gfCNCPoint3[28774] = {X 352.3341, Y -3.5325, Z 11.0000, A 0.000, B 0.000, C 0.000 }
gfCNCPoint3[28775] = {X 352.3341, Y -3.5325, Z -1.6667, A 0.000, B 0.000, C 0.000 }
gfCNCPoint3[28776] = {X 352.3341, Y -3.5325, Z -4.6667, A 0.000, B 0.000, C 0.000 }
gfCNCPoint3[28777] = {X 351.5863, Y 0.4784, Z -4.6667, A 0.000, B 0.000, C 0.000 }
gfCNCPoint3[28778] = {X 351.8700, Y 0.5313, Z -4.6667, A 0.000, B 0.000, C 0.000 }
gfCNCPoint3[28779] = {X 353.8050, Y 1.0172, Z -4.6667, A 0.000, B 0.000, C 0.000 }
gfCNCPoint3[28780] = {X 355.6853, Y 1.6845, Z -4.6667, A 0.000, B 0.000, C 0.000 }
gfCNCPoint3[28781] = {X 357.4938, Y 2.5269, Z -4.6667, A 0.000, B 0.000, C 0.000 }
gfCNCPoint3[28782] = {X 359.2143, Y 3.5371, Z -4.6667, A 0.000, B 0.000, C 0.000 }
gfCNCPoint3[28783] = {X 360.8312, Y 4.7058, Z -4.6667, A 0.000, B 0.000, C 0.000 }
gfCNCPoint3[28784] = {X 362.3301, Y 6.0226, Z -4.6667, A 0.000, B 0.000, C 0.000 }
gfCNCPoint3[28785] = {X 363.6974, Y 7.4756, Z -4.6667, A 0.000, B 0.000, C 0.000 }
gfCNCPoint3[28786] = {X 365.1619, Y 9.3656, Z -4.6667, A 0.000, B 0.000, C 0.000 }
gfCNCPoint3[28787] = {X 366.4369, Y 11.3883, Z -4.6667, A 0.000, B 0.000, C 0.000 }
gfCNCPoint3[28788] = {X 367.5105, Y 13.5247, Z -4.6667, A 0.000, B 0.000, C 0.000 }
gfCNCPoint3[28789] = {X 368.3726, Y 15.7549, Z -4.6667, A 0.000, B 0.000, C 0.000 }
gfCNCPoint3[28790] = {X 369.0153, Y 18.0579, Z -4.6667, A 0.000, B 0.000, C 0.000 }
gfCNCPoint3[28791] = {X 369.4989, Y 20.6961, Z -4.6667, A 0.000, B 0.000, C 0.000 }
gfCNCPoint3[28792] = {X 369.7571, Y 23.3657, Z -4.6667, A 0.000, B 0.000, C 0.000 }
gfCNCPoint3[28793] = {X 369.7880, Y 26.0477, Z -4.6667, A 0.000, B 0.000, C 0.000 }
gfCNCPoint3[28794] = {X 369.5915, Y 28.7226, Z -4.6667, A 0.000, B 0.000, C 0.000 }
gfCNCPoint3[28795] = {X 369.1690, Y 31.3712, Z -4.6667, A 0.000, B 0.000, C 0.000 }
gfCNCPoint3[28796] = {X 368.6451, Y 33.4755, Z -4.6667, A 0.000, B 0.000, C 0.000 }
gfCNCPoint3[28797] = {X 367.9373, Y 35.5252, Z -4.6667, A 0.000, B 0.000, C 0.000 }
gfCNCPoint3[28798] = {X 367.0512, Y 37.5044, Z -4.6667, A 0.000, B 0.000, C 0.000 }
gfCNCPoint3[28799] = {X 365.9938, Y 39.3976, Z -4.6667, A 0.000, B 0.000, C 0.000 }
gfCNCPoint3[28800] = {X 364.7733, Y 41.1900, Z -4.6667, A 0.000, B 0.000, C 0.000 }
gfCNCPoint3[28801] = {X 364.6545, Y 41.3528, Z -4.6667, A 0.000, B 0.000, C 0.000 }
gfCNCPoint3[28802] = {X 364.0247, Y 42.1261, Z -4.6667, A 0.000, B 0.000, C 0.000 }
gfCNCPoint3[28803] = {X 362.7636, Y 43.5412, Z -4.6667, A 0.000, B 0.000, C 0.000 }
gfCNCPoint3[28804] = {X 361.3817, Y 44.8384, Z -4.6667, A 0.000, B 0.000, C 0.000 }
gfCNCPoint3[28805] = {X 359.8899, Y 46.0077, Z -4.6667, A 0.000, B 0.000, C 0.000 }
gfCNCPoint3[28806] = {X 358.3000, Y 47.0398, Z -4.6667, A 0.000, B 0.000, C 0.000 }
gfCNCPoint3[28807] = {X 356.6247, Y 47.9264, Z -4.6667, A 0.000, B 0.000, C 0.000 }
gfCNCPoint3[28808] = {X 356.2232, Y 48.1165, Z -4.6667, A 0.000, B 0.000, C 0.000 }
gfCNCPoint3[28809] = {X 354.0252, Y 48.9371, Z -4.6667, A 0.000, B 0.000, C 0.000 }
gfCNCPoint3[28810] = {X 351.7551, Y 49.5298, Z -4.6667, A 0.000, B 0.000, C 0.000 }
gfCNCPoint3[28811] = {X 349.4364, Y 49.8883, Z -4.6667, A 0.000, B 0.000, C 0.000 }
gfCNCPoint3[28812] = {X 347.0933, Y 50.0089, Z -4.6667, A 0.000, B 0.000, C 0.000 }
gfCNCPoint3[28813] = {X 345.0267, Y 49.9741, Z -4.6667, A 0.000, B 0.000, C 0.000 }
gfCNCPoint3[28814] = {X 342.9709, Y 49.7601, Z -4.6667, A 0.000, B 0.000, C 0.000 }
gfCNCPoint3[28815] = {X 340.9414, Y 49.3687, Z -4.6667, A 0.000, B 0.000, C 0.000 }
gfCNCPoint3[28816] = {X 338.9535, Y 48.8027, Z -4.6667, A 0.000, B 0.000, C 0.000 }
gfCNCPoint3[28817] = {X 337.0223, Y 48.0664, Z -4.6667, A 0.000, B 0.000, C 0.000 }
gfCNCPoint3[28818] = {X 335.1621, Y 47.1654, Z -4.6667, A 0.000, B 0.000, C 0.000 }
gfCNCPoint3[28819] = {X 333.5779, Y 46.1879, Z -4.6667, A 0.000, B 0.000, C 0.000 }
gfCNCPoint3[28820] = {X 332.0749, Y 45.0895, Z -4.6667, A 0.000, B 0.000, C 0.000 }
gfCNCPoint3[28821] = {X 330.6624, Y 43.8770, Z -4.6667, A 0.000, B 0.000, C 0.000 }
gfCNCPoint3[28822] = {X 329.7213, Y 43.8764, Z -4.6667, A 0.000, B 0.000, C 0.000 }
gfCNCPoint3[28823] = {X 328.8027, Y 43.6721, Z -4.6667, A 0.000, B 0.000, C 0.000 }
gfCNCPoint3[28824] = {X 327.9501, Y 43.2738, Z -4.6667, A 0.000, B 0.000, C 0.000 }
gfCNCPoint3[28825] = {X 327.2040, Y 42.7002, Z -4.6667, A 0.000, B 0.000, C 0.000 }
gfCNCPoint3[28826] = {X 326.5808, Y 42.0925, Z -4.6667, A 0.000, B 0.000, C 0.000 }
gfCNCPoint3[28827] = {X 325.9523, Y 41.3190, Z -4.6667, A 0.000, B 0.000, C 0.000 }
gfCNCPoint3[28828] = {X 325.5179, Y 40.4220, Z -4.6667, A 0.000, B 0.000, C 0.000 }
gfCNCPoint3[28829] = {X 325.3006, Y 39.4493, Z -4.6667, A 0.000, B 0.000, C 0.000 }
gfCNCPoint3[28830] = {X 325.3120, Y 38.4527, Z -4.6667, A 0.000, B 0.000, C 0.000 }
gfCNCPoint3[28831] = {X 325.5514, Y 37.4852, Z -4.6667, A 0.000, B 0.000, C 0.000 }
gfCNCPoint3[28832] = {X 326.0062, Y 36.5984, Z -4.6667, A 0.000, B 0.000, C 0.000 }
gfCNCPoint3[28833] = {X 330.2395, Y 30.2687, Z -4.6667, A 0.000, B 0.000, C 0.000 }
gfCNCPoint3[28834] = {X 330.8410, Y 29.5518, Z -4.6667, A 0.000, B 0.000, C 0.000 }
gfCNCPoint3[28835] = {X 331.5827, Y 28.9812, Z -4.6667, A 0.000, B 0.000, C 0.000 }
gfCNCPoint3[28836] = {X 332.4298, Y 28.5837, Z -4.6667, A 0.000, B 0.000, C 0.000 }
gfCNCPoint3[28837] = {X 333.3427, Y 28.3779, Z -4.6667, A 0.000, B 0.000, C 0.000 }
gfCNCPoint3[28838] = {X 334.2785, Y 28.3736, Z -4.6667, A 0.000, B 0.000, C 0.000 }
gfCNCPoint3[28839] = {X 335.1933, Y 28.5709, Z -4.6667, A 0.000, B 0.000, C 0.000 }
gfCNCPoint3[28840] = {X 336.0441, Y 28.9606, Z -4.6667, A 0.000, B 0.000, C 0.000 }
gfCNCPoint3[28841] = {X 336.7910, Y 29.5243, Z -4.6667, A 0.000, B 0.000, C 0.000 }
gfCNCPoint3[28842] = {X 337.4284, Y 30.1382, Z -4.6667, A 0.000, B 0.000, C 0.000 }
gfCNCPoint3[28843] = {X 337.9529, Y 30.7612, Z -4.6667, A 0.000, B 0.000, C 0.000 }
gfCNCPoint3[28844] = {X 338.3512, Y 31.4715, Z -4.6667, A 0.000, B 0.000, C 0.000 }
gfCNCPoint3[28845] = {X 338.6091, Y 32.2439, Z -4.6667, A 0.000, B 0.000, C 0.000 }
gfCNCPoint3[28846] = {X 338.7175, Y 33.0510, Z -4.6667, A 0.000, B 0.000, C 0.000 }
gfCNCPoint3[28847] = {X 338.6725, Y 33.8642, Z -4.6667, A 0.000, B 0.000, C 0.000 }
gfCNCPoint3[28848] = {X 339.4371, Y 34.5550, Z -4.6667, A 0.000, B 0.000, C 0.000 }
gfCNCPoint3[28849] = {X 340.2341, Y 35.2082, Z -4.6667, A 0.000, B 0.000, C 0.000 }
gfCNCPoint3[28850] = {X 341.5315, Y 36.0599, Z -4.6667, A 0.000, B 0.000, C 0.000 }
gfCNCPoint3[28851] = {X 342.9391, Y 36.7134, Z -4.6667, A 0.000, B 0.000, C 0.000 }
gfCNCPoint3[28852] = {X 344.4270, Y 37.1548, Z -4.6667, A 0.000, B 0.000, C 0.000 }
gfCNCPoint3[28853] = {X 345.9633, Y 37.3746, Z -4.6667, A 0.000, B 0.000, C 0.000 }
gfCNCPoint3[28854] = {X 347.5152, Y 37.3683, Z -4.6667, A 0.000, B 0.000, C 0.000 }
gfCNCPoint3[28855] = {X 348.9560, Y 37.1753, Z -4.6667, A 0.000, B 0.000, C 0.000 }
gfCNCPoint3[28856] = {X 350.3462, Y 36.7501, Z -4.6667, A 0.000, B 0.000, C 0.000 }
gfCNCPoint3[28857] = {X 351.6486, Y 36.1043, Z -4.6667, A 0.000, B 0.000, C 0.000 }
gfCNCPoint3[28858] = {X 352.8283, Y 35.2549, Z -4.6667, A 0.000, B 0.000, C 0.000 }
gfCNCPoint3[28859] = {X 353.9821, Y 34.1341, Z -4.6667, A 0.000, B 0.000, C 0.000 }
gfCNCPoint3[28860] = {X 354.9806, Y 32.8730, Z -4.6667, A 0.000, B 0.000, C 0.000 }
gfCNCPoint3[28861] = {X 355.8069, Y 31.4930, Z -4.6667, A 0.000, B 0.000, C 0.000 }
gfCNCPoint3[28862] = {X 356.4470, Y 30.0173, Z -4.6667, A 0.000, B 0.000, C 0.000 }
gfCNCPoint3[28863] = {X 356.8901, Y 28.4711, Z -4.6667, A 0.000, B 0.000, C 0.000 }
gfCNCPoint3[28864] = {X 357.1634, Y 26.7828, Z -4.6667, A 0.000, B 0.000, C 0.000 }
gfCNCPoint3[28865] = {X 357.2747, Y 25.0763, Z -4.6667, A 0.000, B 0.000, C 0.000 }
gfCNCPoint3[28866] = {X 357.2231, Y 23.3669, Z -4.6667, A 0.000, B 0.000, C 0.000 }
gfCNCPoint3[28867] = {X 357.0089, Y 21.6701, Z -4.6667, A 0.000, B 0.000, C 0.000 }
gfCNCPoint3[28868] = {X 356.6550, Y 20.1540, Z -4.6667, A 0.000, B 0.000, C 0.000 }
gfCNCPoint3[28869] = {X 356.1053, Y 18.6975, Z -4.6667, A 0.000, B 0.000, C 0.000 }
gfCNCPoint3[28870] = {X 355.3691, Y 17.3257, Z -4.6667, A 0.000, B 0.000, C 0.000 }
gfCNCPoint3[28871] = {X 354.4594, Y 16.0623, Z -4.6667, A 0.000, B 0.000, C 0.000 }
gfCNCPoint3[28872] = {X 353.5887, Y 15.1354, Z -4.6667, A 0.000, B 0.000, C 0.000 }
gfCNCPoint3[28873] = {X 352.5980, Y 14.3381, Z -4.6667, A 0.000, B 0.000, C 0.000 }
gfCNCPoint3[28874] = {X 351.5062, Y 13.6859, Z -4.6667, A 0.000, B 0.000, C 0.000 }
gfCNCPoint3[28875] = {X 350.3346, Y 13.1914, Z -4.6667, A 0.000, B 0.000, C 0.000 }
gfCNCPoint3[28876] = {X 349.1057, Y 12.8640, Z -4.6667, A 0.000, B 0.000, C 0.000 }
gfCNCPoint3[28877] = {X 347.3453, Y 12.6451, Z -4.6667, A 0.000, B 0.000, C 0.000 }
gfCNCPoint3[28878] = {X 345.5714, Y 12.6609, Z -4.6667, A 0.000, B 0.000, C 0.000 }
gfCNCPoint3[28879] = {X 343.8152, Y 12.9112, Z -4.6667, A 0.000, B 0.000, C 0.000 }
gfCNCPoint3[28880] = {X 342.1076, Y 13.3916, Z -4.6667, A 0.000, B 0.000, C 0.000 }
gfCNCPoint3[28881] = {X 340.4785, Y 14.0937, Z -4.6667, A 0.000, B 0.000, C 0.000 }
gfCNCPoint3[28882] = {X 338.9566, Y 15.0051, Z -4.6667, A 0.000, B 0.000, C 0.000 }
gfCNCPoint3[28883] = {X 338.9177, Y 15.8498, Z -4.6667, A 0.000, B 0.000, C 0.000 }
gfCNCPoint3[28884] = {X 338.7151, Y 16.6708, Z -4.6667, A 0.000, B 0.000, C 0.000 }
gfCNCPoint3[28885] = {X 338.3564, Y 17.4366, Z -4.6667, A 0.000, B 0.000, C 0.000 }
gfCNCPoint3[28886] = {X 337.8553, Y 18.1179, Z -4.6667, A 0.000, B 0.000, C 0.000 }
gfCNCPoint3[28887] = {X 337.2312, Y 18.6884, Z -4.6667, A 0.000, B 0.000, C 0.000 }
gfCNCPoint3[28888] = {X 336.5140, Y 19.2162, Z -4.6667, A 0.000, B 0.000, C 0.000 }
gfCNCPoint3[28889] = {X 335.6982, Y 19.6754, Z -4.6667, A 0.000, B 0.000, C 0.000 }
gfCNCPoint3[28890] = {X 334.8027, Y 19.9480, Z -4.6667, A 0.000, B 0.000, C 0.000 }
gfCNCPoint3[28891] = {X 333.8694, Y 20.0213, Z -4.6667, A 0.000, B 0.000, C 0.000 }
gfCNCPoint3[28892] = {X 332.9422, Y 19.8919, Z -4.6667, A 0.000, B 0.000, C 0.000 }
gfCNCPoint3[28893] = {X 332.0647, Y 19.5657, Z -4.6667, A 0.000, B 0.000, C 0.000 }
gfCNCPoint3[28894] = {X 331.2781, Y 19.0581, Z -4.6667, A 0.000, B 0.000, C 0.000 }
gfCNCPoint3[28895] = {X 330.6193, Y 18.3931, Z -4.6667, A 0.000, B 0.000, C 0.000 }
gfCNCPoint3[28896] = {X 330.1192, Y 17.6017, Z -4.6667, A 0.000, B 0.000, C 0.000 }
gfCNCPoint3[28897] = {X 326.5942, Y 10.3502, Z -4.6667, A 0.000, B 0.000, C 0.000 }
gfCNCPoint3[28898] = {X 326.2930, Y 9.5272, Z -4.6667, A 0.000, B 0.000, C 0.000 }
gfCNCPoint3[28899] = {X 326.1640, Y 8.6602, Z -4.6667, A 0.000, B 0.000, C 0.000 }
gfCNCPoint3[28900] = {X 326.2128, Y 7.7851, Z -4.6667, A 0.000, B 0.000, C 0.000 }
gfCNCPoint3[28901] = {X 326.4371, Y 6.9379, Z -4.6667, A 0.000, B 0.000, C 0.000 }
gfCNCPoint3[28902] = {X 326.8278, Y 6.1534, Z -4.6667, A 0.000, B 0.000, C 0.000 }
gfCNCPoint3[28903] = {X 327.3688, Y 5.4638, Z -4.6667, A 0.000, B 0.000, C 0.000 }
gfCNCPoint3[28904] = {X 328.0379, Y 4.8977, Z -4.6667, A 0.000, B 0.000, C 0.000 }
gfCNCPoint3[28905] = {X 328.7084, Y 4.4386, Z -4.6667, A 0.000, B 0.000, C 0.000 }
gfCNCPoint3[28906] = {X 329.5888, Y 3.9825, Z -4.6667, A 0.000, B 0.000, C 0.000 }
gfCNCPoint3[28907] = {X 330.5501, Y 3.7392, Z -4.6667, A 0.000, B 0.000, C 0.000 }
gfCNCPoint3[28908] = {X 331.5414, Y 3.7215, Z -4.6667, A 0.000, B 0.000, C 0.000 }
gfCNCPoint3[28909] = {X 332.5107, Y 3.9303, Z -4.6667, A 0.000, B 0.000, C 0.000 }
gfCNCPoint3[28910] = {X 333.9976, Y 3.1006, Z -4.6667, A 0.000, B 0.000, C 0.000 }
gfCNCPoint3[28911] = {X 335.5315, Y 2.3616, Z -4.6667, A 0.000, B 0.000, C 0.000 }
gfCNCPoint3[28912] = {X 337.6677, Y 1.4950, Z -4.6667, A 0.000, B 0.000, C 0.000 }
gfCNCPoint3[28913] = {X 339.8716, Y 0.8189, Z -4.6667, A 0.000, B 0.000, C 0.000 }
gfCNCPoint3[28914] = {X 342.1263, Y 0.3386, Z -4.6667, A 0.000, B 0.000, C 0.000 }
gfCNCPoint3[28915] = {X 344.4144, Y 0.0577, Z -4.6667, A 0.000, B 0.000, C 0.000 }
gfCNCPoint3[28916] = {X 346.7183, Y -0.0216, Z -4.6667, A 0.000, B 0.000, C 0.000 }
gfCNCPoint3[28917] = {X 349.0203, Y 0.1013, Z -4.6667, A 0.000, B 0.000, C 0.000 }
gfCNCPoint3[28918] = {X 351.3027, Y 0.4255, Z -4.6667, A 0.000, B 0.000, C 0.000 }
gfCNCPoint3[28919] = {X 351.5863, Y 0.4784, Z -4.6667, A 0.000, B 0.000, C 0.000 }
gfCNCPoint3[28920] = {X 352.3195, Y -3.4539, Z -4.6667, A 0.000, B 0.000, C 0.000 }
gfCNCPoint3[28921] = {X 351.5717, Y 0.5570, Z -4.6667, A 0.000, B 0.000, C 0.000 }
gfCNCPoint3[28922] = {X 351.8548, Y 0.6098, Z -4.6667, A 0.000, B 0.000, C 0.000 }
gfCNCPoint3[28923] = {X 353.7823, Y 1.0939, Z -4.6667, A 0.000, B 0.000, C 0.000 }
gfCNCPoint3[28924] = {X 355.6553, Y 1.7586, Z -4.6667, A 0.000, B 0.000, C 0.000 }
gfCNCPoint3[28925] = {X 357.4569, Y 2.5979, Z -4.6667, A 0.000, B 0.000, C 0.000 }
gfCNCPoint3[28926] = {X 359.1708, Y 3.6042, Z -4.6667, A 0.000, B 0.000, C 0.000 }
gfCNCPoint3[28927] = {X 360.7815, Y 4.7685, Z -4.6667, A 0.000, B 0.000, C 0.000 }
gfCNCPoint3[28928] = {X 362.2746, Y 6.0802, Z -4.6667, A 0.000, B 0.000, C 0.000 }
gfCNCPoint3[28929] = {X 363.6366, Y 7.5276, Z -4.6667, A 0.000, B 0.000, C 0.000 }
gfCNCPoint3[28930] = {X 365.0963, Y 9.4115, Z -4.6667, A 0.000, B 0.000, C 0.000 }
gfCNCPoint3[28931] = {X 366.3672, Y 11.4276, Z -4.6667, A 0.000, B 0.000, C 0.000 }
gfCNCPoint3[28932] = {X 367.4374, Y 13.5571, Z -4.6667, A 0.000, B 0.000, C 0.000 }
gfCNCPoint3[28933] = {X 368.2967, Y 15.7801, Z -4.6667, A 0.000, B 0.000, C 0.000 }
gfCNCPoint3[28934] = {X 368.9373, Y 18.0757, Z -4.6667, A 0.000, B 0.000, C 0.000 }
gfCNCPoint3[28935] = {X 369.4196, Y 20.7071, Z -4.6667, A 0.000, B 0.000, C 0.000 }
gfCNCPoint3[28936] = {X 369.6772, Y 23.3700, Z -4.6667, A 0.000, B 0.000, C 0.000 }
gfCNCPoint3[28937] = {X 369.7081, Y 26.0452, Z -4.6667, A 0.000, B 0.000, C 0.000 }
gfCNCPoint3[28938] = {X 369.5121, Y 28.7133, Z -4.6667, A 0.000, B 0.000, C 0.000 }
gfCNCPoint3[28939] = {X 369.0906, Y 31.3552, Z -4.6667, A 0.000, B 0.000, C 0.000 }
gfCNCPoint3[28940] = {X 368.5684, Y 33.4527, Z -4.6667, A 0.000, B 0.000, C 0.000 }
gfCNCPoint3[28941] = {X 367.8629, Y 35.4959, Z -4.6667, A 0.000, B 0.000, C 0.000 }
gfCNCPoint3[28942] = {X 366.9796, Y 37.4688, Z -4.6667, A 0.000, B 0.000, C 0.000 }
gfCNCPoint3[28943] = {X 365.9256, Y 39.3559, Z -4.6667, A 0.000, B 0.000, C 0.000 }
gfCNCPoint3[28944] = {X 364.7089, Y 41.1425, Z -4.6667, A 0.000, B 0.000, C 0.000 }
gfCNCPoint3[28945] = {X 364.5911, Y 41.3039, Z -4.6667, A 0.000, B 0.000, C 0.000 }
gfCNCPoint3[28946] = {X 363.9627, Y 42.0756, Z -4.6667, A 0.000, B 0.000, C 0.000 }
gfCNCPoint3[28947] = {X 362.7063, Y 43.4853, Z -4.6667, A 0.000, B 0.000, C 0.000 }
gfCNCPoint3[28948] = {X 361.3296, Y 44.7777, Z -4.6667, A 0.000, B 0.000, C 0.000 }
gfCNCPoint3[28949] = {X 359.8434, Y 45.9426, Z -4.6667, A 0.000, B 0.000, C 0.000 }
gfCNCPoint3[28950] = {X 358.2595, Y 46.9708, Z -4.6667, A 0.000, B 0.000, C 0.000 }
gfCNCPoint3[28951] = {X 356.5905, Y 47.8541, Z -4.6667, A 0.000, B 0.000, C 0.000 }
gfCNCPoint3[28952] = {X 356.1902, Y 48.0436, Z -4.6667, A 0.000, B 0.000, C 0.000 }
gfCNCPoint3[28953] = {X 353.9998, Y 48.8612, Z -4.6667, A 0.000, B 0.000, C 0.000 }
gfCNCPoint3[28954] = {X 351.7376, Y 49.4517, Z -4.6667, A 0.000, B 0.000, C 0.000 }
gfCNCPoint3[28955] = {X 349.4271, Y 49.8088, Z -4.6667, A 0.000, B 0.000, C 0.000 }
gfCNCPoint3[28956] = {X 347.0922, Y 49.9289, Z -4.6667, A 0.000, B 0.000, C 0.000 }
gfCNCPoint3[28957] = {X 345.0325, Y 49.8943, Z -4.6667, A 0.000, B 0.000, C 0.000 }
gfCNCPoint3[28958] = {X 342.9836, Y 49.6811, Z -4.6667, A 0.000, B 0.000, C 0.000 }
gfCNCPoint3[28959] = {X 340.9608, Y 49.2911, Z -4.6667, A 0.000, B 0.000, C 0.000 }
gfCNCPoint3[28960] = {X 338.9796, Y 48.7270, Z -4.6667, A 0.000, B 0.000, C 0.000 }
gfCNCPoint3[28961] = {X 337.0547, Y 47.9933, Z -4.6667, A 0.000, B 0.000, C 0.000 }
gfCNCPoint3[28962] = {X 335.2008, Y 47.0953, Z -4.6667, A 0.000, B 0.000, C 0.000 }
gfCNCPoint3[28963] = {X 333.6119, Y 46.1143, Z -4.6667, A 0.000, B 0.000, C 0.000 }
gfCNCPoint3[28964] = {X 332.1052, Y 45.0114, Z -4.6667, A 0.000, B 0.000, C 0.000 }
gfCNCPoint3[28965] = {X 330.6899, Y 43.7933, Z -4.6667, A 0.000, B 0.000, C 0.000 }
gfCNCPoint3[28966] = {X 329.7572, Y 43.7998, Z -4.6667, A 0.000, B 0.000, C 0.000 }
gfCNCPoint3[28967] = {X 328.8457, Y 43.6022, Z -4.6667, A 0.000, B 0.000, C 0.000 }
gfCNCPoint3[28968] = {X 327.9994, Y 43.2101, Z -4.6667, A 0.000, B 0.000, C 0.000 }
gfCNCPoint3[28969] = {X 327.2594, Y 42.6425, Z -4.6667, A 0.000, B 0.000, C 0.000 }
gfCNCPoint3[28970] = {X 326.6366, Y 42.0352, Z -4.6667, A 0.000, B 0.000, C 0.000 }
gfCNCPoint3[28971] = {X 326.0198, Y 41.2760, Z -4.6667, A 0.000, B 0.000, C 0.000 }
gfCNCPoint3[28972] = {X 325.5934, Y 40.3956, Z -4.6667, A 0.000, B 0.000, C 0.000 }
gfCNCPoint3[28973] = {X 325.3802, Y 39.4410, Z -4.6667, A 0.000, B 0.000, C 0.000 }
gfCNCPoint3[28974] = {X 325.3913, Y 38.4628, Z -4.6667, A 0.000, B 0.000, C 0.000 }
gfCNCPoint3[28975] = {X 325.6264, Y 37.5133, Z -4.6667, A 0.000, B 0.000, C 0.000 }
gfCNCPoint3[28976] = {X 326.0727, Y 36.6429, Z -4.6667, A 0.000, B 0.000, C 0.000 }
gfCNCPoint3[28977] = {X 330.3060, Y 30.3132, Z -4.6667, A 0.000, B 0.000, C 0.000 }
gfCNCPoint3[28978] = {X 330.8963, Y 29.6095, Z -4.6667, A 0.000, B 0.000, C 0.000 }
gfCNCPoint3[28979] = {X 331.6243, Y 29.0495, Z -4.6667, A 0.000, B 0.000, C 0.000 }
gfCNCPoint3[28980] = {X 332.4558, Y 28.6594, Z -4.6667, A 0.000, B 0.000, C 0.000 }
gfCNCPoint3[28981] = {X 333.3518, Y 28.4574, Z -4.6667, A 0.000, B 0.000, C 0.000 }
gfCNCPoint3[28982] = {X 334.2702, Y 28.4532, Z -4.6667, A 0.000, B 0.000, C 0.000 }
gfCNCPoint3[28983] = {X 335.1680, Y 28.6468, Z -4.6667, A 0.000, B 0.000, C 0.000 }
gfCNCPoint3[28984] = {X 336.0031, Y 29.0293, Z -4.6667, A 0.000, B 0.000, C 0.000 }
gfCNCPoint3[28985] = {X 336.7362, Y 29.5826, Z -4.6667, A 0.000, B 0.000, C 0.000 }
gfCNCPoint3[28986] = {X 337.3723, Y 30.1953, Z -4.6667, A 0.000, B 0.000, C 0.000 }
gfCNCPoint3[28987] = {X 337.8919, Y 30.8135, Z -4.6667, A 0.000, B 0.000, C 0.000 }
gfCNCPoint3[28988] = {X 338.2848, Y 31.5191, Z -4.6667, A 0.000, B 0.000, C 0.000 }
gfCNCPoint3[28989] = {X 338.5368, Y 32.2863, Z -4.6667, A 0.000, B 0.000, C 0.000 }
gfCNCPoint3[28990] = {X 338.6387, Y 33.0874, Z -4.6667, A 0.000, B 0.000, C 0.000 }
gfCNCPoint3[28991] = {X 338.5870, Y 33.8933, Z -4.6667, A 0.000, B 0.000, C 0.000 }
gfCNCPoint3[28992] = {X 339.3691, Y 34.6020, Z -4.6667, A 0.000, B 0.000, C 0.000 }
gfCNCPoint3[28993] = {X 340.1851, Y 35.2715, Z -4.6667, A 0.000, B 0.000, C 0.000 }
gfCNCPoint3[28994] = {X 341.4921, Y 36.1296, Z -4.6667, A 0.000, B 0.000, C 0.000 }
gfCNCPoint3[28995] = {X 342.9102, Y 36.7880, Z -4.6667, A 0.000, B 0.000, C 0.000 }
gfCNCPoint3[28996] = {X 344.4091, Y 37.2328, Z -4.6667, A 0.000, B 0.000, C 0.000 }
gfCNCPoint3[28997] = {X 345.9568, Y 37.4544, Z -4.6667, A 0.000, B 0.000, C 0.000 }
gfCNCPoint3[28998] = {X 347.5203, Y 37.4481, Z -4.6667, A 0.000, B 0.000, C 0.000 }
gfCNCPoint3[28999] = {X 348.6860, Y 37.3112, Z -4.6667, A 0.000, B 0.000, C 0.000 }
gfCNCPoint3[29000] = {X 349.8239, Y 37.0234, Z -4.6667, A 0.000, B 0.000, C 0.000 }
gfCNCPoint3[29001] = {X 350.9144, Y 36.5895, Z -4.6667, A 0.000, B 0.000, C 0.000 }
gfCNCPoint3[29002] = {X 351.9391, Y 36.0170, Z -4.6667, A 0.000, B 0.000, C 0.000 }
gfCNCPoint3[29003] = {X 352.8802, Y 35.3158, Z -4.6667, A 0.000, B 0.000, C 0.000 }
gfCNCPoint3[29004] = {X 354.0415, Y 34.1877, Z -4.6667, A 0.000, B 0.000, C 0.000 }
gfCNCPoint3[29005] = {X 355.0464, Y 32.9184, Z -4.6667, A 0.000, B 0.000, C 0.000 }
gfCNCPoint3[29006] = {X 355.8781, Y 31.5294, Z -4.6667, A 0.000, B 0.000, C 0.000 }
gfCNCPoint3[29007] = {X 356.5224, Y 30.0442, Z -4.6667, A 0.000, B 0.000, C 0.000 }
gfCNCPoint3[29008] = {X 356.9684, Y 28.4878, Z -4.6667, A 0.000, B 0.000, C 0.000 }
gfCNCPoint3[29009] = {X 357.2429, Y 26.7920, Z -4.6667, A 0.000, B 0.000, C 0.000 }
gfCNCPoint3[29010] = {X 357.3547, Y 25.0778, Z -4.6667, A 0.000, B 0.000, C 0.000 }
gfCNCPoint3[29011] = {X 357.3028, Y 23.3607, Z -4.6667, A 0.000, B 0.000, C 0.000 }
gfCNCPoint3[29012] = {X 357.0877, Y 21.6563, Z -4.6667, A 0.000, B 0.000, C 0.000 }
gfCNCPoint3[29013] = {X 356.7314, Y 20.1302, Z -4.6667, A 0.000, B 0.000, C 0.000 }
gfCNCPoint3[29014] = {X 356.1779, Y 18.6640, Z -4.6667, A 0.000, B 0.000, C 0.000 }
gfCNCPoint3[29015] = {X 355.4369, Y 17.2831, Z -4.6667, A 0.000, B 0.000, C 0.000 }
gfCNCPoint3[29016] = {X 354.5211, Y 16.0114, Z -4.6667, A 0.000, B 0.000, C 0.000 }
gfCNCPoint3[29017] = {X 353.6428, Y 15.0764, Z -4.6667, A 0.000, B 0.000, C 0.000 }
gfCNCPoint3[29018] = {X 352.6434, Y 14.2723, Z -4.6667, A 0.000, B 0.000, C 0.000 }
gfCNCPoint3[29019] = {X 351.5422, Y 13.6145, Z -4.6667, A 0.000, B 0.000, C 0.000 }
gfCNCPoint3[29020] = {X 350.3604, Y 13.1156, Z -4.6667, A 0.000, B 0.000, C 0.000 }
gfCNCPoint3[29021] = {X 349.1209, Y 12.7855, Z -4.6667, A 0.000, B 0.000, C 0.000 }
gfCNCPoint3[29022] = {X 347.3425, Y 12.5648, Z -4.6667, A 0.000, B 0.000, C 0.000 }
gfCNCPoint3[29023] = {X 345.5505, Y 12.5823, Z -4.6667, A 0.000, B 0.000, C 0.000 }
gfCNCPoint3[29024] = {X 343.7768, Y 12.8376, Z -4.6667, A 0.000, B 0.000, C 0.000 }
gfCNCPoint3[29025] = {X 342.0527, Y 13.3263, Z -4.6667, A 0.000, B 0.000, C 0.000 }
gfCNCPoint3[29026] = {X 340.4088, Y 14.0396, Z -4.6667, A 0.000, B 0.000, C 0.000 }
gfCNCPoint3[29027] = {X 338.8741, Y 14.9650, Z -4.6667, A 0.000, B 0.000, C 0.000 }
gfCNCPoint3[29028] = {X 338.8435, Y 15.8032, Z -4.6667, A 0.000, B 0.000, C 0.000 }
gfCNCPoint3[29029] = {X 338.6485, Y 16.6190, Z -4.6667, A 0.000, B 0.000, C 0.000 }
gfCNCPoint3[29030] = {X 338.2966, Y 17.3805, Z -4.6667, A 0.000, B 0.000, C 0.000 }
gfCNCPoint3[29031] = {X 337.8018, Y 18.0578, Z -4.6667, A 0.000, B 0.000, C 0.000 }
gfCNCPoint3[29032] = {X 337.1833, Y 18.6244, Z -4.6667, A 0.000, B 0.000, C 0.000 }
gfCNCPoint3[29033] = {X 336.4675, Y 19.1512, Z -4.6667, A 0.000, B 0.000, C 0.000 }
gfCNCPoint3[29034] = {X 335.6668, Y 19.6018, Z -4.6667, A 0.000, B 0.000, C 0.000 }
gfCNCPoint3[29035] = {X 334.7878, Y 19.8694, Z -4.6667, A 0.000, B 0.000, C 0.000 }
gfCNCPoint3[29036] = {X 333.8718, Y 19.9414, Z -4.6667, A 0.000, B 0.000, C 0.000 }
gfCNCPoint3[29037] = {X 332.9618, Y 19.8143, Z -4.6667, A 0.000, B 0.000, C 0.000 }
gfCNCPoint3[29038] = {X 332.1006, Y 19.4942, Z -4.6667, A 0.000, B 0.000, C 0.000 }
gfCNCPoint3[29039] = {X 331.3285, Y 18.9960, Z -4.6667, A 0.000, B 0.000, C 0.000 }
gfCNCPoint3[29040] = {X 330.6819, Y 18.3433, Z -4.6667, A 0.000, B 0.000, C 0.000 }
gfCNCPoint3[29041] = {X 330.1911, Y 17.5665, Z -4.6667, A 0.000, B 0.000, C 0.000 }
gfCNCPoint3[29042] = {X 326.6662, Y 10.3152, Z -4.6667, A 0.000, B 0.000, C 0.000 }
gfCNCPoint3[29043] = {X 326.3374, Y 9.3677, Z -4.6667, A 0.000, B 0.000, C 0.000 }
gfCNCPoint3[29044] = {X 326.2405, Y 8.3694, Z -4.6667, A 0.000, B 0.000, C 0.000 }
gfCNCPoint3[29045] = {X 326.3807, Y 7.3763, Z -4.6667, A 0.000, B 0.000, C 0.000 }
gfCNCPoint3[29046] = {X 326.7503, Y 6.4439, Z -4.6667, A 0.000, B 0.000, C 0.000 }
gfCNCPoint3[29047] = {X 327.3286, Y 5.6244, Z -4.6667, A 0.000, B 0.000, C 0.000 }
gfCNCPoint3[29048] = {X 328.0831, Y 4.9637, Z -4.6667, A 0.000, B 0.000, C 0.000 }
gfCNCPoint3[29049] = {X 328.7533, Y 4.5047, Z -4.6667, A 0.000, B 0.000, C 0.000 }
gfCNCPoint3[29050] = {X 329.6261, Y 4.0539, Z -4.6667, A 0.000, B 0.000, C 0.000 }
gfCNCPoint3[29051] = {X 330.5791, Y 3.8161, Z -4.6667, A 0.000, B 0.000, C 0.000 }
gfCNCPoint3[29052] = {X 331.5613, Y 3.8039, Z -4.6667, A 0.000, B 0.000, C 0.000 }
gfCNCPoint3[29053] = {X 332.5199, Y 4.0180, Z -4.6667, A 0.000, B 0.000, C 0.000 }
gfCNCPoint3[29054] = {X 334.0181, Y 3.1800, Z -4.6667, A 0.000, B 0.000, C 0.000 }
gfCNCPoint3[29055] = {X 335.5645, Y 2.4345, Z -4.6667, A 0.000, B 0.000, C 0.000 }
gfCNCPoint3[29056] = {X 337.6942, Y 1.5705, Z -4.6667, A 0.000, B 0.000, C 0.000 }
gfCNCPoint3[29057] = {X 339.8914, Y 0.8965, Z -4.6667, A 0.000, B 0.000, C 0.000 }
gfCNCPoint3[29058] = {X 342.1393, Y 0.4176, Z -4.6667, A 0.000, B 0.000, C 0.000 }
gfCNCPoint3[29059] = {X 344.4205, Y 0.1375, Z -4.6667, A 0.000, B 0.000, C 0.000 }
gfCNCPoint3[29060] = {X 346.7174, Y 0.0584, Z -4.6667, A 0.000, B 0.000, C 0.000 }
gfCNCPoint3[29061] = {X 349.0125, Y 0.1810, Z -4.6667, A 0.000, B 0.000, C 0.000 }
gfCNCPoint3[29062] = {X 351.2879, Y 0.5041, Z -4.6667, A 0.000, B 0.000, C 0.000 }
gfCNCPoint3[29063] = {X 351.5717, Y 0.5570, Z -4.6667, A 0.000, B 0.000, C 0.000 }
gfCNCPoint3[29064] = {X 352.3048, Y -3.3752, Z -4.6667, A 0.000, B 0.000, C 0.000 }
gfCNCPoint3[29065] = {X 351.5570, Y 0.6357, Z -4.6667, A 0.000, B 0.000, C 0.000 }
gfCNCPoint3[29066] = {X 351.8395, Y 0.6884, Z -4.6667, A 0.000, B 0.000, C 0.000 }
gfCNCPoint3[29067] = {X 353.7597, Y 1.1707, Z -4.6667, A 0.000, B 0.000, C 0.000 }
gfCNCPoint3[29068] = {X 355.6254, Y 1.8328, Z -4.6667, A 0.000, B 0.000, C 0.000 }
gfCNCPoint3[29069] = {X 357.4200, Y 2.6689, Z -4.6667, A 0.000, B 0.000, C 0.000 }
gfCNCPoint3[29070] = {X 359.1272, Y 3.6714, Z -4.6667, A 0.000, B 0.000, C 0.000 }
gfCNCPoint3[29071] = {X 360.7317, Y 4.8311, Z -4.6667, A 0.000, B 0.000, C 0.000 }
gfCNCPoint3[29072] = {X 362.2190, Y 6.1378, Z -4.6667, A 0.000, B 0.000, C 0.000 }
gfCNCPoint3[29073] = {X 363.5758, Y 7.5796, Z -4.6667, A 0.000, B 0.000, C 0.000 }
gfCNCPoint3[29074] = {X 365.0308, Y 9.4574, Z -4.6667, A 0.000, B 0.000, C 0.000 }
gfCNCPoint3[29075] = {X 366.2976, Y 11.4670, Z -4.6667, A 0.000, B 0.000, C 0.000 }
gfCNCPoint3[29076] = {X 367.3642, Y 13.5896, Z -4.6667, A 0.000, B 0.000, C 0.000 }
gfCNCPoint3[29077] = {X 368.2208, Y 15.8053, Z -4.6667, A 0.000, B 0.000, C 0.000 }
gfCNCPoint3[29078] = {X 368.8593, Y 18.0934, Z -4.6667, A 0.000, B 0.000, C 0.000 }
gfCNCPoint3[29079] = {X 369.3404, Y 20.7182, Z -4.6667, A 0.000, B 0.000, C 0.000 }
gfCNCPoint3[29080] = {X 369.5973, Y 23.3744, Z -4.6667, A 0.000, B 0.000, C 0.000 }
gfCNCPoint3[29081] = {X 369.6281, Y 26.0427, Z -4.6667, A 0.000, B 0.000, C 0.000 }
gfCNCPoint3[29082] = {X 369.4326, Y 28.7041, Z -4.6667, A 0.000, B 0.000, C 0.000 }
gfCNCPoint3[29083] = {X 369.0122, Y 31.3393, Z -4.6667, A 0.000, B 0.000, C 0.000 }
gfCNCPoint3[29084] = {X 368.4916, Y 33.4300, Z -4.6667, A 0.000, B 0.000, C 0.000 }
gfCNCPoint3[29085] = {X 367.7884, Y 35.4666, Z -4.6667, A 0.000, B 0.000, C 0.000 }
gfCNCPoint3[29086] = {X 366.9080, Y 37.4331, Z -4.6667, A 0.000, B 0.000, C 0.000 }
gfCNCPoint3[29087] = {X 365.8573, Y 39.3141, Z -4.6667, A 0.000, B 0.000, C 0.000 }
gfCNCPoint3[29088] = {X 364.6446, Y 41.0949, Z -4.6667, A 0.000, B 0.000, C 0.000 }
gfCNCPoint3[29089] = {X 364.5278, Y 41.2551, Z -4.6667, A 0.000, B 0.000, C 0.000 }
gfCNCPoint3[29090] = {X 363.9006, Y 42.0251, Z -4.6667, A 0.000, B 0.000, C 0.000 }
gfCNCPoint3[29091] = {X 362.6490, Y 43.4295, Z -4.6667, A 0.000, B 0.000, C 0.000 }
gfCNCPoint3[29092] = {X 361.2774, Y 44.7170, Z -4.6667, A 0.000, B 0.000, C 0.000 }
gfCNCPoint3[29093] = {X 359.7969, Y 45.8775, Z -4.6667, A 0.000, B 0.000, C 0.000 }
gfCNCPoint3[29094] = {X 358.2190, Y 46.9018, Z -4.6667, A 0.000, B 0.000, C 0.000 }
gfCNCPoint3[29095] = {X 356.5563, Y 47.7818, Z -4.6667, A 0.000, B 0.000, C 0.000 }
gfCNCPoint3[29096] = {X 356.1572, Y 47.9707, Z -4.6667, A 0.000, B 0.000, C 0.000 }
gfCNCPoint3[29097] = {X 353.9745, Y 48.7853, Z -4.6667, A 0.000, B 0.000, C 0.000 }
gfCNCPoint3[29098] = {X 351.7202, Y 49.3736, Z -4.6667, A 0.000, B 0.000, C 0.000 }
gfCNCPoint3[29099] = {X 349.4178, Y 49.7293, Z -4.6667, A 0.000, B 0.000, C 0.000 }
gfCNCPoint3[29100] = {X 347.0911, Y 49.8489, Z -4.6667, A 0.000, B 0.000, C 0.000 }
gfCNCPoint3[29101] = {X 345.0383, Y 49.8145, Z -4.6667, A 0.000, B 0.000, C 0.000 }
gfCNCPoint3[29102] = {X 342.9962, Y 49.6022, Z -4.6667, A 0.000, B 0.000, C 0.000 }
gfCNCPoint3[29103] = {X 340.9803, Y 49.2135, Z -4.6667, A 0.000, B 0.000, C 0.000 }
gfCNCPoint3[29104] = {X 339.0056, Y 48.6514, Z -4.6667, A 0.000, B 0.000, C 0.000 }
gfCNCPoint3[29105] = {X 337.0872, Y 47.9202, Z -4.6667, A 0.000, B 0.000, C 0.000 }
gfCNCPoint3[29106] = {X 335.2394, Y 47.0253, Z -4.6667, A 0.000, B 0.000, C 0.000 }
gfCNCPoint3[29107] = {X 333.6459, Y 46.0408, Z -4.6667, A 0.000, B 0.000, C 0.000 }
gfCNCPoint3[29108] = {X 332.1353, Y 44.9332, Z -4.6667, A 0.000, B 0.000, C 0.000 }
gfCNCPoint3[29109] = {X 330.7172, Y 43.7094, Z -4.6667, A 0.000, B 0.000, C 0.000 }
gfCNCPoint3[29110] = {X 329.7931, Y 43.7230, Z -4.6667, A 0.000, B 0.000, C 0.000 }
gfCNCPoint3[29111] = {X 328.8887, Y 43.5322, Z -4.6667, A 0.000, B 0.000, C 0.000 }
gfCNCPoint3[29112] = {X 328.0488, Y 43.1464, Z -4.6667, A 0.000, B 0.000, C 0.000 }
gfCNCPoint3[29113] = {X 327.3148, Y 42.5847, Z -4.6667, A 0.000, B 0.000, C 0.000 }
gfCNCPoint3[29114] = {X 326.6925, Y 41.9780, Z -4.6667, A 0.000, B 0.000, C 0.000 }
gfCNCPoint3[29115] = {X 326.0873, Y 41.2331, Z -4.6667, A 0.000, B 0.000, C 0.000 }
gfCNCPoint3[29116] = {X 325.6690, Y 40.3693, Z -4.6667, A 0.000, B 0.000, C 0.000 }
gfCNCPoint3[29117] = {X 325.4597, Y 39.4326, Z -4.6667, A 0.000, B 0.000, C 0.000 }
gfCNCPoint3[29118] = {X 325.4707, Y 38.4730, Z -4.6667, A 0.000, B 0.000, C 0.000 }
gfCNCPoint3[29119] = {X 325.7013, Y 37.5413, Z -4.6667, A 0.000, B 0.000, C 0.000 }
gfCNCPoint3[29120] = {X 326.1392, Y 36.6874, Z -4.6667, A 0.000, B 0.000, C 0.000 }
gfCNCPoint3[29121] = {X 330.3725, Y 30.3576, Z -4.6667, A 0.000, B 0.000, C 0.000 }
gfCNCPoint3[29122] = {X 330.9516, Y 29.6673, Z -4.6667, A 0.000, B 0.000, C 0.000 }
gfCNCPoint3[29123] = {X 331.6658, Y 29.1179, Z -4.6667, A 0.000, B 0.000, C 0.000 }
gfCNCPoint3[29124] = {X 332.4816, Y 28.7351, Z -4.6667, A 0.000, B 0.000, C 0.000 }
gfCNCPoint3[29125] = {X 333.3606, Y 28.5370, Z -4.6667, A 0.000, B 0.000, C 0.000 }
gfCNCPoint3[29126] = {X 334.2616, Y 28.5327, Z -4.6667, A 0.000, B 0.000, C 0.000 }
gfCNCPoint3[29127] = {X 335.1425, Y 28.7227, Z -4.6667, A 0.000, B 0.000, C 0.000 }
gfCNCPoint3[29128] = {X 335.9617, Y 29.0978, Z -4.6667, A 0.000, B 0.000, C 0.000 }
gfCNCPoint3[29129] = {X 336.6810, Y 29.6405, Z -4.6667, A 0.000, B 0.000, C 0.000 }
gfCNCPoint3[29130] = {X 337.3163, Y 30.2523, Z -4.6667, A 0.000, B 0.000, C 0.000 }
gfCNCPoint3[29131] = {X 337.8308, Y 30.8658, Z -4.6667, A 0.000, B 0.000, C 0.000 }
gfCNCPoint3[29132] = {X 338.2182, Y 31.5665, Z -4.6667, A 0.000, B 0.000, C 0.000 }
gfCNCPoint3[29133] = {X 338.4642, Y 32.3285, Z -4.6667, A 0.000, B 0.000, C 0.000 }
gfCNCPoint3[29134] = {X 338.5597, Y 33.1234, Z -4.6667, A 0.000, B 0.000, C 0.000 }
gfCNCPoint3[29135] = {X 338.5011, Y 33.9219, Z -4.6667, A 0.000, B 0.000, C 0.000 }
gfCNCPoint3[29136] = {X 339.3009, Y 34.6489, Z -4.6667, A 0.000, B 0.000, C 0.000 }
gfCNCPoint3[29137] = {X 340.1361, Y 35.3348, Z -4.6667, A 0.000, B 0.000, C 0.000 }
gfCNCPoint3[29138] = {X 341.4528, Y 36.1992, Z -4.6667, A 0.000, B 0.000, C 0.000 }
gfCNCPoint3[29139] = {X 342.8813, Y 36.8626, Z -4.6667, A 0.000, B 0.000, C 0.000 }
gfCNCPoint3[29140] = {X 344.3913, Y 37.3108, Z -4.6667, A 0.000, B 0.000, C 0.000 }
gfCNCPoint3[29141] = {X 345.9504, Y 37.5341, Z -4.6667, A 0.000, B 0.000, C 0.000 }
gfCNCPoint3[29142] = {X 347.5255, Y 37.5280, Z -4.6667, A 0.000, B 0.000, C 0.000 }
gfCNCPoint3[29143] = {X 348.7013, Y 37.3897, Z -4.6667, A 0.000, B 0.000, C 0.000 }
gfCNCPoint3[29144] = {X 349.8491, Y 37.0993, Z -4.6667, A 0.000, B 0.000, C 0.000 }
gfCNCPoint3[29145] = {X 350.9492, Y 36.6616, Z -4.6667, A 0.000, B 0.000, C 0.000 }
gfCNCPoint3[29146] = {X 351.9827, Y 36.0841, Z -4.6667, A 0.000, B 0.000, C 0.000 }
gfCNCPoint3[29147] = {X 352.9321, Y 35.3766, Z -4.6667, A 0.000, B 0.000, C 0.000 }
gfCNCPoint3[29148] = {X 354.1009, Y 34.2413, Z -4.6667, A 0.000, B 0.000, C 0.000 }
gfCNCPoint3[29149] = {X 355.1123, Y 32.9638, Z -4.6667, A 0.000, B 0.000, C 0.000 }
gfCNCPoint3[29150] = {X 355.9493, Y 31.5658, Z -4.6667, A 0.000, B 0.000, C 0.000 }
gfCNCPoint3[29151] = {X 356.5978, Y 30.0710, Z -4.6667, A 0.000, B 0.000, C 0.000 }
gfCNCPoint3[29152] = {X 357.0466, Y 28.5046, Z -4.6667, A 0.000, B 0.000, C 0.000 }
gfCNCPoint3[29153] = {X 357.3224, Y 26.8012, Z -4.6667, A 0.000, B 0.000, C 0.000 }
gfCNCPoint3[29154] = {X 357.4347, Y 25.0793, Z -4.6667, A 0.000, B 0.000, C 0.000 }
gfCNCPoint3[29155] = {X 357.3826, Y 23.3545, Z -4.6667, A 0.000, B 0.000, C 0.000 }
gfCNCPoint3[29156] = {X 357.1665, Y 21.6425, Z -4.6667, A 0.000, B 0.000, C 0.000 }
gfCNCPoint3[29157] = {X 356.8077, Y 20.1064, Z -4.6667, A 0.000, B 0.000, C 0.000 }
gfCNCPoint3[29158] = {X 356.2506, Y 18.6306, Z -4.6667, A 0.000, B 0.000, C 0.000 }
gfCNCPoint3[29159] = {X 355.5046, Y 17.2406, Z -4.6667, A 0.000, B 0.000, C 0.000 }
gfCNCPoint3[29160] = {X 354.5828, Y 15.9605, Z -4.6667, A 0.000, B 0.000, C 0.000 }
gfCNCPoint3[29161] = {X 353.6970, Y 15.0175, Z -4.6667, A 0.000, B 0.000, C 0.000 }
gfCNCPoint3[29162] = {X 352.6889, Y 14.2065, Z -4.6667, A 0.000, B 0.000, C 0.000 }
gfCNCPoint3[29163] = {X 351.5782, Y 13.5430, Z -4.6667, A 0.000, B 0.000, C 0.000 }
gfCNCPoint3[29164] = {X 350.3862, Y 13.0399, Z -4.6667, A 0.000, B 0.000, C 0.000 }
gfCNCPoint3[29165] = {X 349.1360, Y 12.7069, Z -4.6667, A 0.000, B 0.000, C 0.000 }
gfCNCPoint3[29166] = {X 347.5978, Y 12.5015, Z -4.6667, A 0.000, B 0.000, C 0.000 }
gfCNCPoint3[29167] = {X 346.0461, Y 12.4735, Z -4.6667, A 0.000, B 0.000, C 0.000 }
gfCNCPoint3[29168] = {X 344.5014, Y 12.6231, Z -4.6667, A 0.000, B 0.000, C 0.000 }
gfCNCPoint3[29169] = {X 342.9840, Y 12.9485, Z -4.6667, A 0.000, B 0.000, C 0.000 }
gfCNCPoint3[29170] = {X 341.5138, Y 13.4454, Z -4.6667, A 0.000, B 0.000, C 0.000 }
gfCNCPoint3[29171] = {X 340.1100, Y 14.1072, Z -4.6667, A 0.000, B 0.000, C 0.000 }
gfCNCPoint3[29172] = {X 338.7913, Y 14.9253, Z -4.6667, A 0.000, B 0.000, C 0.000 }
gfCNCPoint3[29173] = {X 338.7689, Y 15.7569, Z -4.6667, A 0.000, B 0.000, C 0.000 }
gfCNCPoint3[29174] = {X 338.5816, Y 16.5674, Z -4.6667, A 0.000, B 0.000, C 0.000 }
gfCNCPoint3[29175] = {X 338.2367, Y 17.3245, Z -4.6667, A 0.000, B 0.000, C 0.000 }
gfCNCPoint3[29176] = {X 337.7481, Y 17.9978, Z -4.6667, A 0.000, B 0.000, C 0.000 }
gfCNCPoint3[29177] = {X 337.1353, Y 18.5604, Z -4.6667, A 0.000, B 0.000, C 0.000 }
gfCNCPoint3[29178] = {X 336.4209, Y 19.0861, Z -4.6667, A 0.000, B 0.000, C 0.000 }
gfCNCPoint3[29179] = {X 335.6353, Y 19.5283, Z -4.6667, A 0.000, B 0.000, C 0.000 }
gfCNCPoint3[29180] = {X 334.7729, Y 19.7908, Z -4.6667, A 0.000, B 0.000, C 0.000 }
gfCNCPoint3[29181] = {X 333.8742, Y 19.8614, Z -4.6667, A 0.000, B 0.000, C 0.000 }
gfCNCPoint3[29182] = {X 332.9814, Y 19.7367, Z -4.6667, A 0.000, B 0.000, C 0.000 }
gfCNCPoint3[29183] = {X 332.1364, Y 19.4226, Z -4.6667, A 0.000, B 0.000, C 0.000 }
gfCNCPoint3[29184] = {X 331.3789, Y 18.9339, Z -4.6667, A 0.000, B 0.000, C 0.000 }
gfCNCPoint3[29185] = {X 330.7445, Y 18.2934, Z -4.6667, A 0.000, B 0.000, C 0.000 }
gfCNCPoint3[29186] = {X 330.2630, Y 17.5314, Z -4.6667, A 0.000, B 0.000, C 0.000 }
gfCNCPoint3[29187] = {X 326.7381, Y 10.2803, Z -4.6667, A 0.000, B 0.000, C 0.000 }
gfCNCPoint3[29188] = {X 326.4156, Y 9.3506, Z -4.6667, A 0.000, B 0.000, C 0.000 }
gfCNCPoint3[29189] = {X 326.3205, Y 8.3711, Z -4.6667, A 0.000, B 0.000, C 0.000 }
gfCNCPoint3[29190] = {X 326.4580, Y 7.3968, Z -4.6667, A 0.000, B 0.000, C 0.000 }
gfCNCPoint3[29191] = {X 326.8207, Y 6.4820, Z -4.6667, A 0.000, B 0.000, C 0.000 }
gfCNCPoint3[29192] = {X 327.3880, Y 5.6779, Z -4.6667, A 0.000, B 0.000, C 0.000 }
gfCNCPoint3[29193] = {X 328.1283, Y 5.0297, Z -4.6667, A 0.000, B 0.000, C 0.000 }
gfCNCPoint3[29194] = {X 328.7983, Y 4.5709, Z -4.6667, A 0.000, B 0.000, C 0.000 }
gfCNCPoint3[29195] = {X 329.6632, Y 4.1254, Z -4.6667, A 0.000, B 0.000, C 0.000 }
gfCNCPoint3[29196] = {X 330.6080, Y 3.8930, Z -4.6667, A 0.000, B 0.000, C 0.000 }
gfCNCPoint3[29197] = {X 331.5809, Y 3.8865, Z -4.6667, A 0.000, B 0.000, C 0.000 }
gfCNCPoint3[29198] = {X 332.5288, Y 4.1060, Z -4.6667, A 0.000, B 0.000, C 0.000 }
gfCNCPoint3[29199] = {X 334.0385, Y 3.2596, Z -4.6667, A 0.000, B 0.000, C 0.000 }
gfCNCPoint3[29200] = {X 335.5974, Y 2.5074, Z -4.6667, A 0.000, B 0.000, C 0.000 }
gfCNCPoint3[29201] = {X 337.7207, Y 1.6460, Z -4.6667, A 0.000, B 0.000, C 0.000 }
gfCNCPoint3[29202] = {X 339.9113, Y 0.9740, Z -4.6667, A 0.000, B 0.000, C 0.000 }
gfCNCPoint3[29203] = {X 342.1523, Y 0.4965, Z -4.6667, A 0.000, B 0.000, C 0.000 }
gfCNCPoint3[29204] = {X 344.4266, Y 0.2173, Z -4.6667, A 0.000, B 0.000, C 0.000 }
gfCNCPoint3[29205] = {X 346.7166, Y 0.1384, Z -4.6667, A 0.000, B 0.000, C 0.000 }
gfCNCPoint3[29206] = {X 349.0047, Y 0.2606, Z -4.6667, A 0.000, B 0.000, C 0.000 }
gfCNCPoint3[29207] = {X 351.2732, Y 0.5828, Z -4.6667, A 0.000, B 0.000, C 0.000 }
gfCNCPoint3[29208] = {X 351.5570, Y 0.6357, Z -4.6667, A 0.000, B 0.000, C 0.000 }
gfCNCPoint3[29209] = {X 352.2901, Y -3.2966, Z -4.6667, A 0.000, B 0.000, C 0.000 }
gfCNCPoint3[29210] = {X 352.2902, Y -3.2966, Z -4.6667, A 0.000, B 0.000, C 0.000 }
gfCNCPoint3[29211] = {X 351.5423, Y 0.7143, Z -4.6667, A 0.000, B 0.000, C 0.000 }
gfCNCPoint3[29212] = {X 351.8243, Y 0.7669, Z -4.6667, A 0.000, B 0.000, C 0.000 }
gfCNCPoint3[29213] = {X 353.7370, Y 1.2474, Z -4.6667, A 0.000, B 0.000, C 0.000 }
gfCNCPoint3[29214] = {X 355.5955, Y 1.9070, Z -4.6667, A 0.000, B 0.000, C 0.000 }
gfCNCPoint3[29215] = {X 357.3831, Y 2.7399, Z -4.6667, A 0.000, B 0.000, C 0.000 }
gfCNCPoint3[29216] = {X 359.0837, Y 3.7385, Z -4.6667, A 0.000, B 0.000, C 0.000 }
gfCNCPoint3[29217] = {X 360.6820, Y 4.8938, Z -4.6667, A 0.000, B 0.000, C 0.000 }
gfCNCPoint3[29218] = {X 362.1635, Y 6.1954, Z -4.6667, A 0.000, B 0.000, C 0.000 }
gfCNCPoint3[29219] = {X 363.5150, Y 7.6316, Z -4.6667, A 0.000, B 0.000, C 0.000 }
gfCNCPoint3[29220] = {X 364.9653, Y 9.5033, Z -4.6667, A 0.000, B 0.000, C 0.000 }
gfCNCPoint3[29221] = {X 366.2279, Y 11.5063, Z -4.6667, A 0.000, B 0.000, C 0.000 }
gfCNCPoint3[29222] = {X 367.2911, Y 13.6220, Z -4.6667, A 0.000, B 0.000, C 0.000 }
gfCNCPoint3[29223] = {X 368.1449, Y 15.8305, Z -4.6667, A 0.000, B 0.000, C 0.000 }
gfCNCPoint3[29224] = {X 368.7813, Y 18.1112, Z -4.6667, A 0.000, B 0.000, C 0.000 }
gfCNCPoint3[29225] = {X 369.2612, Y 20.7293, Z -4.6667, A 0.000, B 0.000, C 0.000 }
gfCNCPoint3[29226] = {X 369.5174, Y 23.3787, Z -4.6667, A 0.000, B 0.000, C 0.000 }
gfCNCPoint3[29227] = {X 369.5482, Y 26.0403, Z -4.6667, A 0.000, B 0.000, C 0.000 }
gfCNCPoint3[29228] = {X 369.3531, Y 28.6948, Z -4.6667, A 0.000, B 0.000, C 0.000 }
gfCNCPoint3[29229] = {X 368.9338, Y 31.3234, Z -4.6667, A 0.000, B 0.000, C 0.000 }
gfCNCPoint3[29230] = {X 368.4149, Y 33.4073, Z -4.6667, A 0.000, B 0.000, C 0.000 }
gfCNCPoint3[29231] = {X 367.7140, Y 35.4373, Z -4.6667, A 0.000, B 0.000, C 0.000 }
gfCNCPoint3[29232] = {X 366.8364, Y 37.3974, Z -4.6667, A 0.000, B 0.000, C 0.000 }
gfCNCPoint3[29233] = {X 365.7891, Y 39.2723, Z -4.6667, A 0.000, B 0.000, C 0.000 }
gfCNCPoint3[29234] = {X 364.5802, Y 41.0474, Z -4.6667, A 0.000, B 0.000, C 0.000 }
gfCNCPoint3[29235] = {X 364.4644, Y 41.2062, Z -4.6667, A 0.000, B 0.000, C 0.000 }
gfCNCPoint3[29236] = {X 363.8386, Y 41.9746, Z -4.6667, A 0.000, B 0.000, C 0.000 }
gfCNCPoint3[29237] = {X 362.5917, Y 43.3737, Z -4.6667, A 0.000, B 0.000, C 0.000 }
gfCNCPoint3[29238] = {X 361.2253, Y 44.6563, Z -4.6667, A 0.000, B 0.000, C 0.000 }
gfCNCPoint3[29239] = {X 359.7504, Y 45.8124, Z -4.6667, A 0.000, B 0.000, C 0.000 }
gfCNCPoint3[29240] = {X 358.1784, Y 46.8328, Z -4.6667, A 0.000, B 0.000, C 0.000 }
gfCNCPoint3[29241] = {X 356.5220, Y 47.7095, Z -4.6667, A 0.000, B 0.000, C 0.000 }
gfCNCPoint3[29242] = {X 356.1242, Y 47.8978, Z -4.6667, A 0.000, B 0.000, C 0.000 }
gfCNCPoint3[29243] = {X 353.9492, Y 48.7094, Z -4.6667, A 0.000, B 0.000, C 0.000 }
gfCNCPoint3[29244] = {X 351.7028, Y 49.2955, Z -4.6667, A 0.000, B 0.000, C 0.000 }
gfCNCPoint3[29245] = {X 349.4085, Y 49.6499, Z -4.6667, A 0.000, B 0.000, C 0.000 }
gfCNCPoint3[29246] = {X 347.0900, Y 49.7689, Z -4.6667, A 0.000, B 0.000, C 0.000 }
gfCNCPoint3[29247] = {X 345.0441, Y 49.7347, Z -4.6667, A 0.000, B 0.000, C 0.000 }
gfCNCPoint3[29248] = {X 343.0089, Y 49.5232, Z -4.6667, A 0.000, B 0.000, C 0.000 }
gfCNCPoint3[29249] = {X 340.9997, Y 49.1359, Z -4.6667, A 0.000, B 0.000, C 0.000 }
gfCNCPoint3[29250] = {X 339.0317, Y 48.5757, Z -4.6667, A 0.000, B 0.000, C 0.000 }
gfCNCPoint3[29251] = {X 337.1196, Y 47.8470, Z -4.6667, A 0.000, B 0.000, C 0.000 }
gfCNCPoint3[29252] = {X 335.2780, Y 46.9552, Z -4.6667, A 0.000, B 0.000, C 0.000 }
gfCNCPoint3[29253] = {X 333.6797, Y 45.9671, Z -4.6667, A 0.000, B 0.000, C 0.000 }
gfCNCPoint3[29254] = {X 332.1653, Y 44.8547, Z -4.6667, A 0.000, B 0.000, C 0.000 }
gfCNCPoint3[29255] = {X 330.7443, Y 43.6252, Z -4.6667, A 0.000, B 0.000, C 0.000 }
gfCNCPoint3[29256] = {X 329.8287, Y 43.6460, Z -4.6667, A 0.000, B 0.000, C 0.000 }
gfCNCPoint3[29257] = {X 328.9316, Y 43.4621, Z -4.6667, A 0.000, B 0.000, C 0.000 }
gfCNCPoint3[29258] = {X 328.0980, Y 43.0827, Z -4.6667, A 0.000, B 0.000, C 0.000 }
gfCNCPoint3[29259] = {X 327.3701, Y 42.5270, Z -4.6667, A 0.000, B 0.000, C 0.000 }
gfCNCPoint3[29260] = {X 326.7483, Y 41.9207, Z -4.6667, A 0.000, B 0.000, C 0.000 }
gfCNCPoint3[29261] = {X 326.1548, Y 41.1901, Z -4.6667, A 0.000, B 0.000, C 0.000 }
gfCNCPoint3[29262] = {X 325.7445, Y 40.3430, Z -4.6667, A 0.000, B 0.000, C 0.000 }
gfCNCPoint3[29263] = {X 325.5393, Y 39.4243, Z -4.6667, A 0.000, B 0.000, C 0.000 }
gfCNCPoint3[29264] = {X 325.5500, Y 38.4831, Z -4.6667, A 0.000, B 0.000, C 0.000 }
gfCNCPoint3[29265] = {X 325.7762, Y 37.5694, Z -4.6667, A 0.000, B 0.000, C 0.000 }
gfCNCPoint3[29266] = {X 326.2057, Y 36.7318, Z -4.6667, A 0.000, B 0.000, C 0.000 }
gfCNCPoint3[29267] = {X 330.4390, Y 30.4021, Z -4.6667, A 0.000, B 0.000, C 0.000 }
gfCNCPoint3[29268] = {X 331.0070, Y 29.7251, Z -4.6667, A 0.000, B 0.000, C 0.000 }
gfCNCPoint3[29269] = {X 331.7073, Y 29.1862, Z -4.6667, A 0.000, B 0.000, C 0.000 }
gfCNCPoint3[29270] = {X 332.5073, Y 28.8108, Z -4.6667, A 0.000, B 0.000, C 0.000 }
gfCNCPoint3[29271] = {X 333.3694, Y 28.6165, Z -4.6667, A 0.000, B 0.000, C 0.000 }
gfCNCPoint3[29272] = {X 334.2531, Y 28.6123, Z -4.6667, A 0.000, B 0.000, C 0.000 }
gfCNCPoint3[29273] = {X 335.1169, Y 28.7985, Z -4.6667, A 0.000, B 0.000, C 0.000 }
gfCNCPoint3[29274] = {X 335.9204, Y 29.1663, Z -4.6667, A 0.000, B 0.000, C 0.000 }
gfCNCPoint3[29275] = {X 336.6259, Y 29.6985, Z -4.6667, A 0.000, B 0.000, C 0.000 }
gfCNCPoint3[29276] = {X 337.2602, Y 30.3094, Z -4.6667, A 0.000, B 0.000, C 0.000 }
gfCNCPoint3[29277] = {X 337.7696, Y 30.9181, Z -4.6667, A 0.000, B 0.000, C 0.000 }
gfCNCPoint3[29278] = {X 338.1515, Y 31.6139, Z -4.6667, A 0.000, B 0.000, C 0.000 }
gfCNCPoint3[29279] = {X 338.3914, Y 32.3704, Z -4.6667, A 0.000, B 0.000, C 0.000 }
gfCNCPoint3[29280] = {X 338.4804, Y 33.1591, Z -4.6667, A 0.000, B 0.000, C 0.000 }
gfCNCPoint3[29281] = {X 338.4149, Y 33.9501, Z -4.6667, A 0.000, B 0.000, C 0.000 }
gfCNCPoint3[29282] = {X 339.2325, Y 34.6955, Z -4.6667, A 0.000, B 0.000, C 0.000 }
gfCNCPoint3[29283] = {X 340.0872, Y 35.3980, Z -4.6667, A 0.000, B 0.000, C 0.000 }
gfCNCPoint3[29284] = {X 341.4134, Y 36.2689, Z -4.6667, A 0.000, B 0.000, C 0.000 }
gfCNCPoint3[29285] = {X 342.8524, Y 36.9372, Z -4.6667, A 0.000, B 0.000, C 0.000 }
gfCNCPoint3[29286] = {X 344.3734, Y 37.3887, Z -4.6667, A 0.000, B 0.000, C 0.000 }
gfCNCPoint3[29287] = {X 345.9440, Y 37.6139, Z -4.6667, A 0.000, B 0.000, C 0.000 }
gfCNCPoint3[29288] = {X 347.5306, Y 37.6078, Z -4.6667, A 0.000, B 0.000, C 0.000 }
gfCNCPoint3[29289] = {X 348.7167, Y 37.4683, Z -4.6667, A 0.000, B 0.000, C 0.000 }
gfCNCPoint3[29290] = {X 349.8744, Y 37.1752, Z -4.6667, A 0.000, B 0.000, C 0.000 }
gfCNCPoint3[29291] = {X 350.9839, Y 36.7336, Z -4.6667, A 0.000, B 0.000, C 0.000 }
gfCNCPoint3[29292] = {X 352.0264, Y 36.1511, Z -4.6667, A 0.000, B 0.000, C 0.000 }
gfCNCPoint3[29293] = {X 352.9840, Y 35.4375, Z -4.6667, A 0.000, B 0.000, C 0.000 }
gfCNCPoint3[29294] = {X 354.1603, Y 34.2949, Z -4.6667, A 0.000, B 0.000, C 0.000 }
gfCNCPoint3[29295] = {X 355.1782, Y 33.0092, Z -4.6667, A 0.000, B 0.000, C 0.000 }
gfCNCPoint3[29296] = {X 356.0206, Y 31.6022, Z -4.6667, A 0.000, B 0.000, C 0.000 }
gfCNCPoint3[29297] = {X 356.6731, Y 30.0978, Z -4.6667, A 0.000, B 0.000, C 0.000 }
gfCNCPoint3[29298] = {X 357.1248, Y 28.5214, Z -4.6667, A 0.000, B 0.000, C 0.000 }
gfCNCPoint3[29299] = {X 357.4018, Y 26.8104, Z -4.6667, A 0.000, B 0.000, C 0.000 }
gfCNCPoint3[29300] = {X 357.5147, Y 25.0808, Z -4.6667, A 0.000, B 0.000, C 0.000 }
gfCNCPoint3[29301] = {X 357.4624, Y 23.3484, Z -4.6667, A 0.000, B 0.000, C 0.000 }
gfCNCPoint3[29302] = {X 357.2453, Y 21.6288, Z -4.6667, A 0.000, B 0.000, C 0.000 }
gfCNCPoint3[29303] = {X 356.8841, Y 20.0826, Z -4.6667, A 0.000, B 0.000, C 0.000 }
gfCNCPoint3[29304] = {X 356.3232, Y 18.5971, Z -4.6667, A 0.000, B 0.000, C 0.000 }
gfCNCPoint3[29305] = {X 355.5724, Y 17.1981, Z -4.6667, A 0.000, B 0.000, C 0.000 }
gfCNCPoint3[29306] = {X 354.6445, Y 15.9096, Z -4.6667, A 0.000, B 0.000, C 0.000 }
gfCNCPoint3[29307] = {X 353.7511, Y 14.9586, Z -4.6667, A 0.000, B 0.000, C 0.000 }
gfCNCPoint3[29308] = {X 352.7344, Y 14.1407, Z -4.6667, A 0.000, B 0.000, C 0.000 }
gfCNCPoint3[29309] = {X 351.6142, Y 13.4716, Z -4.6667, A 0.000, B 0.000, C 0.000 }
gfCNCPoint3[29310] = {X 350.4121, Y 12.9642, Z -4.6667, A 0.000, B 0.000, C 0.000 }
gfCNCPoint3[29311] = {X 349.1512, Y 12.6284, Z -4.6667, A 0.000, B 0.000, C 0.000 }
gfCNCPoint3[29312] = {X 347.5973, Y 12.4213, Z -4.6667, A 0.000, B 0.000, C 0.000 }
gfCNCPoint3[29313] = {X 346.0299, Y 12.3941, Z -4.6667, A 0.000, B 0.000, C 0.000 }
gfCNCPoint3[29314] = {X 344.4698, Y 12.5471, Z -4.6667, A 0.000, B 0.000, C 0.000 }
gfCNCPoint3[29315] = {X 342.9376, Y 12.8783, Z -4.6667, A 0.000, B 0.000, C 0.000 }
gfCNCPoint3[29316] = {X 341.4536, Y 13.3835, Z -4.6667, A 0.000, B 0.000, C 0.000 }
gfCNCPoint3[29317] = {X 340.0375, Y 14.0557, Z -4.6667, A 0.000, B 0.000, C 0.000 }
gfCNCPoint3[29318] = {X 338.7079, Y 14.8862, Z -4.6667, A 0.000, B 0.000, C 0.000 }
gfCNCPoint3[29319] = {X 338.6940, Y 15.7110, Z -4.6667, A 0.000, B 0.000, C 0.000 }
gfCNCPoint3[29320] = {X 338.5144, Y 16.5161, Z -4.6667, A 0.000, B 0.000, C 0.000 }
gfCNCPoint3[29321] = {X 338.1766, Y 17.2686, Z -4.6667, A 0.000, B 0.000, C 0.000 }
gfCNCPoint3[29322] = {X 337.6944, Y 17.9378, Z -4.6667, A 0.000, B 0.000, C 0.000 }
gfCNCPoint3[29323] = {X 337.0874, Y 18.4963, Z -4.6667, A 0.000, B 0.000, C 0.000 }
gfCNCPoint3[29324] = {X 336.3744, Y 19.0211, Z -4.6667, A 0.000, B 0.000, C 0.000 }
gfCNCPoint3[29325] = {X 335.6039, Y 19.4547, Z -4.6667, A 0.000, B 0.000, C 0.000 }
gfCNCPoint3[29326] = {X 334.7580, Y 19.7122, Z -4.6667, A 0.000, B 0.000, C 0.000 }
gfCNCPoint3[29327] = {X 333.8766, Y 19.7814, Z -4.6667, A 0.000, B 0.000, C 0.000 }
gfCNCPoint3[29328] = {X 333.0010, Y 19.6592, Z -4.6667, A 0.000, B 0.000, C 0.000 }
gfCNCPoint3[29329] = {X 332.1722, Y 19.3511, Z -4.6667, A 0.000, B 0.000, C 0.000 }
gfCNCPoint3[29330] = {X 331.4293, Y 18.8718, Z -4.6667, A 0.000, B 0.000, C 0.000 }
gfCNCPoint3[29331] = {X 330.8071, Y 18.2436, Z -4.6667, A 0.000, B 0.000, C 0.000 }
gfCNCPoint3[29332] = {X 330.3348, Y 17.4962, Z -4.6667, A 0.000, B 0.000, C 0.000 }
gfCNCPoint3[29333] = {X 326.8100, Y 10.2453, Z -4.6667, A 0.000, B 0.000, C 0.000 }
gfCNCPoint3[29334] = {X 326.4937, Y 9.3335, Z -4.6667, A 0.000, B 0.000, C 0.000 }
gfCNCPoint3[29335] = {X 326.4004, Y 8.3729, Z -4.6667, A 0.000, B 0.000, C 0.000 }
gfCNCPoint3[29336] = {X 326.5354, Y 7.4172, Z -4.6667, A 0.000, B 0.000, C 0.000 }
gfCNCPoint3[29337] = {X 326.8910, Y 6.5200, Z -4.6667, A 0.000, B 0.000, C 0.000 }
gfCNCPoint3[29338] = {X 327.4475, Y 5.7315, Z -4.6667, A 0.000, B 0.000, C 0.000 }
gfCNCPoint3[29339] = {X 328.1735, Y 5.0957, Z -4.6667, A 0.000, B 0.000, C 0.000 }
gfCNCPoint3[29340] = {X 328.8432, Y 4.6371, Z -4.6667, A 0.000, B 0.000, C 0.000 }
gfCNCPoint3[29341] = {X 329.7004, Y 4.1970, Z -4.6667, A 0.000, B 0.000, C 0.000 }
gfCNCPoint3[29342] = {X 330.6369, Y 3.9701, Z -4.6667, A 0.000, B 0.000, C 0.000 }
gfCNCPoint3[29343] = {X 331.6004, Y 3.9692, Z -4.6667, A 0.000, B 0.000, C 0.000 }
gfCNCPoint3[29344] = {X 332.5373, Y 4.1943, Z -4.6667, A 0.000, B 0.000, C 0.000 }
gfCNCPoint3[29345] = {X 334.0588, Y 3.3393, Z -4.6667, A 0.000, B 0.000, C 0.000 }
gfCNCPoint3[29346] = {X 335.6304, Y 2.5803, Z -4.6667, A 0.000, B 0.000, C 0.000 }
gfCNCPoint3[29347] = {X 337.7472, Y 1.7215, Z -4.6667, A 0.000, B 0.000, C 0.000 }
gfCNCPoint3[29348] = {X 339.9311, Y 1.0515, Z -4.6667, A 0.000, B 0.000, C 0.000 }
gfCNCPoint3[29349] = {X 342.1653, Y 0.5754, Z -4.6667, A 0.000, B 0.000, C 0.000 }
gfCNCPoint3[29350] = {X 344.4327, Y 0.2970, Z -4.6667, A 0.000, B 0.000, C 0.000 }
gfCNCPoint3[29351] = {X 346.7157, Y 0.2184, Z -4.6667, A 0.000, B 0.000, C 0.000 }
gfCNCPoint3[29352] = {X 348.9968, Y 0.3402, Z -4.6667, A 0.000, B 0.000, C 0.000 }
gfCNCPoint3[29353] = {X 351.2585, Y 0.6614, Z -4.6667, A 0.000, B 0.000, C 0.000 }
gfCNCPoint3[29354] = {X 351.5423, Y 0.7143, Z -4.6667, A 0.000, B 0.000, C 0.000 }
gfCNCPoint3[29355] = {X 352.2755, Y -3.2179, Z -4.6667, A 0.000, B 0.000, C 0.000 }
gfCNCPoint3[29356] = {X 351.5277, Y 0.7930, Z -4.6667, A 0.000, B 0.000, C 0.000 }
gfCNCPoint3[29357] = {X 351.8091, Y 0.8454, Z -4.6667, A 0.000, B 0.000, C 0.000 }
gfCNCPoint3[29358] = {X 353.7143, Y 1.3241, Z -4.6667, A 0.000, B 0.000, C 0.000 }
gfCNCPoint3[29359] = {X 355.5656, Y 1.9812, Z -4.6667, A 0.000, B 0.000, C 0.000 }
gfCNCPoint3[29360] = {X 357.3462, Y 2.8109, Z -4.6667, A 0.000, B 0.000, C 0.000 }
gfCNCPoint3[29361] = {X 359.0402, Y 3.8056, Z -4.6667, A 0.000, B 0.000, C 0.000 }
gfCNCPoint3[29362] = {X 360.6322, Y 4.9564, Z -4.6667, A 0.000, B 0.000, C 0.000 }
gfCNCPoint3[29363] = {X 362.1080, Y 6.2530, Z -4.6667, A 0.000, B 0.000, C 0.000 }
gfCNCPoint3[29364] = {X 363.4542, Y 7.6836, Z -4.6667, A 0.000, B 0.000, C 0.000 }
gfCNCPoint3[29365] = {X 364.8997, Y 9.5491, Z -4.6667, A 0.000, B 0.000, C 0.000 }
gfCNCPoint3[29366] = {X 366.1582, Y 11.5457, Z -4.6667, A 0.000, B 0.000, C 0.000 }
gfCNCPoint3[29367] = {X 367.2179, Y 13.6544, Z -4.6667, A 0.000, B 0.000, C 0.000 }
gfCNCPoint3[29368] = {X 368.0689, Y 15.8557, Z -4.6667, A 0.000, B 0.000, C 0.000 }
gfCNCPoint3[29369] = {X 368.7033, Y 18.1289, Z -4.6667, A 0.000, B 0.000, C 0.000 }
gfCNCPoint3[29370] = {X 369.1819, Y 20.7404, Z -4.6667, A 0.000, B 0.000, C 0.000 }
gfCNCPoint3[29371] = {X 369.4375, Y 23.3830, Z -4.6667, A 0.000, B 0.000, C 0.000 }
gfCNCPoint3[29372] = {X 369.4682, Y 26.0378, Z -4.6667, A 0.000, B 0.000, C 0.000 }
gfCNCPoint3[29373] = {X 369.2737, Y 28.6856, Z -4.6667, A 0.000, B 0.000, C 0.000 }
gfCNCPoint3[29374] = {X 368.8554, Y 31.3074, Z -4.6667, A 0.000, B 0.000, C 0.000 }
gfCNCPoint3[29375] = {X 368.3382, Y 33.3846, Z -4.6667, A 0.000, B 0.000, C 0.000 }
gfCNCPoint3[29376] = {X 367.6395, Y 35.4080, Z -4.6667, A 0.000, B 0.000, C 0.000 }
gfCNCPoint3[29377] = {X 366.7648, Y 37.3618, Z -4.6667, A 0.000, B 0.000, C 0.000 }
gfCNCPoint3[29378] = {X 365.7209, Y 39.2306, Z -4.6667, A 0.000, B 0.000, C 0.000 }
gfCNCPoint3[29379] = {X 364.5159, Y 40.9999, Z -4.6667, A 0.000, B 0.000, C 0.000 }
gfCNCPoint3[29380] = {X 364.4010, Y 41.1573, Z -4.6667, A 0.000, B 0.000, C 0.000 }
gfCNCPoint3[29381] = {X 363.7766, Y 41.9241, Z -4.6667, A 0.000, B 0.000, C 0.000 }
gfCNCPoint3[29382] = {X 362.5344, Y 43.3178, Z -4.6667, A 0.000, B 0.000, C 0.000 }
gfCNCPoint3[29383] = {X 361.1732, Y 44.5956, Z -4.6667, A 0.000, B 0.000, C 0.000 }
gfCNCPoint3[29384] = {X 359.7039, Y 45.7473, Z -4.6667, A 0.000, B 0.000, C 0.000 }
gfCNCPoint3[29385] = {X 358.1379, Y 46.7639, Z -4.6667, A 0.000, B 0.000, C 0.000 }
gfCNCPoint3[29386] = {X 356.4878, Y 47.6371, Z -4.6667, A 0.000, B 0.000, C 0.000 }
gfCNCPoint3[29387] = {X 356.0912, Y 47.8249, Z -4.6667, A 0.000, B 0.000, C 0.000 }
gfCNCPoint3[29388] = {X 353.9238, Y 48.6335, Z -4.6667, A 0.000, B 0.000, C 0.000 }
gfCNCPoint3[29389] = {X 351.6854, Y 49.2174, Z -4.6667, A 0.000, B 0.000, C 0.000 }
gfCNCPoint3[29390] = {X 349.3992, Y 49.5704, Z -4.6667, A 0.000, B 0.000, C 0.000 }
gfCNCPoint3[29391] = {X 347.0889, Y 49.6889, Z -4.6667, A 0.000, B 0.000, C 0.000 }
gfCNCPoint3[29392] = {X 345.0499, Y 49.6549, Z -4.6667, A 0.000, B 0.000, C 0.000 }
gfCNCPoint3[29393] = {X 343.0216, Y 49.4442, Z -4.6667, A 0.000, B 0.000, C 0.000 }
gfCNCPoint3[29394] = {X 341.0191, Y 49.0583, Z -4.6667, A 0.000, B 0.000, C 0.000 }
gfCNCPoint3[29395] = {X 339.0577, Y 48.5001, Z -4.6667, A 0.000, B 0.000, C 0.000 }
gfCNCPoint3[29396] = {X 337.1521, Y 47.7739, Z -4.6667, A 0.000, B 0.000, C 0.000 }
gfCNCPoint3[29397] = {X 335.3167, Y 46.8852, Z -4.6667, A 0.000, B 0.000, C 0.000 }
gfCNCPoint3[29398] = {X 333.7135, Y 45.8934, Z -4.6667, A 0.000, B 0.000, C 0.000 }
gfCNCPoint3[29399] = {X 332.1950, Y 44.7761, Z -4.6667, A 0.000, B 0.000, C 0.000 }
gfCNCPoint3[29400] = {X 330.7711, Y 43.5406, Z -4.6667, A 0.000, B 0.000, C 0.000 }
gfCNCPoint3[29401] = {X 329.8559, Y 43.5681, Z -4.6667, A 0.000, B 0.000, C 0.000 }
gfCNCPoint3[29402] = {X 328.9583, Y 43.3867, Z -4.6667, A 0.000, B 0.000, C 0.000 }
gfCNCPoint3[29403] = {X 328.1256, Y 43.0059, Z -4.6667, A 0.000, B 0.000, C 0.000 }
gfCNCPoint3[29404] = {X 327.4012, Y 42.4458, Z -4.6667, A 0.000, B 0.000, C 0.000 }
gfCNCPoint3[29405] = {X 326.8042, Y 41.8634, Z -4.6667, A 0.000, B 0.000, C 0.000 }
gfCNCPoint3[29406] = {X 326.2223, Y 41.1472, Z -4.6667, A 0.000, B 0.000, C 0.000 }
gfCNCPoint3[29407] = {X 325.8201, Y 40.3166, Z -4.6667, A 0.000, B 0.000, C 0.000 }
gfCNCPoint3[29408] = {X 325.6189, Y 39.4160, Z -4.6667, A 0.000, B 0.000, C 0.000 }
gfCNCPoint3[29409] = {X 325.6294, Y 38.4932, Z -4.6667, A 0.000, B 0.000, C 0.000 }
gfCNCPoint3[29410] = {X 325.8511, Y 37.5974, Z -4.6667, A 0.000, B 0.000, C 0.000 }
gfCNCPoint3[29411] = {X 326.2722, Y 36.7763, Z -4.6667, A 0.000, B 0.000, C 0.000 }
gfCNCPoint3[29412] = {X 330.5290, Y 30.4119, Z -4.6667, A 0.000, B 0.000, C 0.000 }
gfCNCPoint3[29413] = {X 331.0932, Y 29.7536, Z -4.6667, A 0.000, B 0.000, C 0.000 }
gfCNCPoint3[29414] = {X 331.7861, Y 29.2322, Z -4.6667, A 0.000, B 0.000, C 0.000 }
gfCNCPoint3[29415] = {X 332.5750, Y 28.8724, Z -4.6667, A 0.000, B 0.000, C 0.000 }
gfCNCPoint3[29416] = {X 333.4229, Y 28.6911, Z -4.6667, A 0.000, B 0.000, C 0.000 }
gfCNCPoint3[29417] = {X 334.2900, Y 28.6968, Z -4.6667, A 0.000, B 0.000, C 0.000 }
gfCNCPoint3[29418] = {X 335.1355, Y 28.8892, Z -4.6667, A 0.000, B 0.000, C 0.000 }
gfCNCPoint3[29419] = {X 335.9197, Y 29.2593, Z -4.6667, A 0.000, B 0.000, C 0.000 }
gfCNCPoint3[29420] = {X 336.6056, Y 29.7897, Z -4.6667, A 0.000, B 0.000, C 0.000 }
gfCNCPoint3[29421] = {X 337.2041, Y 30.3665, Z -4.6667, A 0.000, B 0.000, C 0.000 }
gfCNCPoint3[29422] = {X 337.7083, Y 30.9703, Z -4.6667, A 0.000, B 0.000, C 0.000 }
gfCNCPoint3[29423] = {X 338.0846, Y 31.6611, Z -4.6667, A 0.000, B 0.000, C 0.000 }
gfCNCPoint3[29424] = {X 338.3184, Y 32.4122, Z -4.6667, A 0.000, B 0.000, C 0.000 }
gfCNCPoint3[29425] = {X 338.4007, Y 33.1945, Z -4.6667, A 0.000, B 0.000, C 0.000 }
gfCNCPoint3[29426] = {X 338.3283, Y 33.9779, Z -4.6667, A 0.000, B 0.000, C 0.000 }
gfCNCPoint3[29427] = {X 339.1639, Y 34.7419, Z -4.6667, A 0.000, B 0.000, C 0.000 }
gfCNCPoint3[29428] = {X 340.0382, Y 35.4613, Z -4.6667, A 0.000, B 0.000, C 0.000 }
gfCNCPoint3[29429] = {X 341.2962, Y 36.2942, Z -4.6667, A 0.000, B 0.000, C 0.000 }
gfCNCPoint3[29430] = {X 342.6568, Y 36.9462, Z -4.6667, A 0.000, B 0.000, C 0.000 }
gfCNCPoint3[29431] = {X 344.0942, Y 37.4048, Z -4.6667, A 0.000, B 0.000, C 0.000 }
gfCNCPoint3[29432] = {X 345.5810, Y 37.6612, Z -4.6667, A 0.000, B 0.000, C 0.000 }
gfCNCPoint3[29433] = {X 347.0889, Y 37.7108, Z -4.6667, A 0.000, B 0.000, C 0.000 }
gfCNCPoint3[29434] = {X 347.5348, Y 37.6877, Z -4.6667, A 0.000, B 0.000, C 0.000 }
gfCNCPoint3[29435] = {X 348.7312, Y 37.5469, Z -4.6667, A 0.000, B 0.000, C 0.000 }
gfCNCPoint3[29436] = {X 349.8990, Y 37.2513, Z -4.6667, A 0.000, B 0.000, C 0.000 }
gfCNCPoint3[29437] = {X 351.0183, Y 36.8059, Z -4.6667, A 0.000, B 0.000, C 0.000 }
gfCNCPoint3[29438] = {X 352.0699, Y 36.2182, Z -4.6667, A 0.000, B 0.000, C 0.000 }
gfCNCPoint3[29439] = {X 353.0359, Y 35.4984, Z -4.6667, A 0.000, B 0.000, C 0.000 }
gfCNCPoint3[29440] = {X 354.2196, Y 34.3485, Z -4.6667, A 0.000, B 0.000, C 0.000 }
gfCNCPoint3[29441] = {X 355.2441, Y 33.0546, Z -4.6667, A 0.000, B 0.000, C 0.000 }
gfCNCPoint3[29442] = {X 356.0918, Y 31.6387, Z -4.6667, A 0.000, B 0.000, C 0.000 }
gfCNCPoint3[29443] = {X 356.7485, Y 30.1246, Z -4.6667, A 0.000, B 0.000, C 0.000 }
gfCNCPoint3[29444] = {X 357.2030, Y 28.5381, Z -4.6667, A 0.000, B 0.000, C 0.000 }
gfCNCPoint3[29445] = {X 357.4813, Y 26.8196, Z -4.6667, A 0.000, B 0.000, C 0.000 }
gfCNCPoint3[29446] = {X 357.5947, Y 25.0823, Z -4.6667, A 0.000, B 0.000, C 0.000 }
gfCNCPoint3[29447] = {X 357.5421, Y 23.3422, Z -4.6667, A 0.000, B 0.000, C 0.000 }
gfCNCPoint3[29448] = {X 357.3241, Y 21.6150, Z -4.6667, A 0.000, B 0.000, C 0.000 }
gfCNCPoint3[29449] = {X 356.9605, Y 20.0587, Z -4.6667, A 0.000, B 0.000, C 0.000 }
gfCNCPoint3[29450] = {X 356.3959, Y 18.5636, Z -4.6667, A 0.000, B 0.000, C 0.000 }
gfCNCPoint3[29451] = {X 355.6401, Y 17.1555, Z -4.6667, A 0.000, B 0.000, C 0.000 }
gfCNCPoint3[29452] = {X 354.7062, Y 15.8586, Z -4.6667, A 0.000, B 0.000, C 0.000 }
gfCNCPoint3[29453] = {X 353.8052, Y 14.8997, Z -4.6667, A 0.000, B 0.000, C 0.000 }
gfCNCPoint3[29454] = {X 352.7799, Y 14.0749, Z -4.6667, A 0.000, B 0.000, C 0.000 }
gfCNCPoint3[29455] = {X 351.6502, Y 13.4001, Z -4.6667, A 0.000, B 0.000, C 0.000 }
gfCNCPoint3[29456] = {X 350.4379, Y 12.8885, Z -4.6667, A 0.000, B 0.000, C 0.000 }
gfCNCPoint3[29457] = {X 349.1664, Y 12.5499, Z -4.6667, A 0.000, B 0.000, C 0.000 }
gfCNCPoint3[29458] = {X 347.3712, Y 12.3261, Z -4.6667, A 0.000, B 0.000, C 0.000 }
gfCNCPoint3[29459] = {X 345.5623, Y 12.3407, Z -4.6667, A 0.000, B 0.000, C 0.000 }
gfCNCPoint3[29460] = {X 343.7710, Y 12.5935, Z -4.6667, A 0.000, B 0.000, C 0.000 }
gfCNCPoint3[29461] = {X 342.0287, Y 13.0801, Z -4.6667, A 0.000, B 0.000, C 0.000 }
gfCNCPoint3[29462] = {X 340.3656, Y 13.7921, Z -4.6667, A 0.000, B 0.000, C 0.000 }
gfCNCPoint3[29463] = {X 338.8108, Y 14.7168, Z -4.6667, A 0.000, B 0.000, C 0.000 }
gfCNCPoint3[29464] = {X 338.7178, Y 14.7814, Z -4.6667, A 0.000, B 0.000, C 0.000 }
gfCNCPoint3[29465] = {X 338.6254, Y 14.8467, Z -4.6667, A 0.000, B 0.000, C 0.000 }
gfCNCPoint3[29466] = {X 338.6379, Y 15.0631, Z -4.6667, A 0.000, B 0.000, C 0.000 }
gfCNCPoint3[29467] = {X 338.5596, Y 16.0356, Z -4.6667, A 0.000, B 0.000, C 0.000 }
gfCNCPoint3[29468] = {X 338.2483, Y 16.9601, Z -4.6667, A 0.000, B 0.000, C 0.000 }
gfCNCPoint3[29469] = {X 337.7224, Y 17.7818, Z -4.6667, A 0.000, B 0.000, C 0.000 }
gfCNCPoint3[29470] = {X 337.0132, Y 18.4517, Z -4.6667, A 0.000, B 0.000, C 0.000 }
gfCNCPoint3[29471] = {X 336.3278, Y 18.9560, Z -4.6667, A 0.000, B 0.000, C 0.000 }
gfCNCPoint3[29472] = {X 335.5713, Y 19.3817, Z -4.6667, A 0.000, B 0.000, C 0.000 }
gfCNCPoint3[29473] = {X 334.7407, Y 19.6341, Z -4.6667, A 0.000, B 0.000, C 0.000 }
gfCNCPoint3[29474] = {X 333.8753, Y 19.7014, Z -4.6667, A 0.000, B 0.000, C 0.000 }
gfCNCPoint3[29475] = {X 333.0157, Y 19.5804, Z -4.6667, A 0.000, B 0.000, C 0.000 }
gfCNCPoint3[29476] = {X 332.2025, Y 19.2768, Z -4.6667, A 0.000, B 0.000, C 0.000 }
gfCNCPoint3[29477] = {X 331.4739, Y 18.8049, Z -4.6667, A 0.000, B 0.000, C 0.000 }
gfCNCPoint3[29478] = {X 330.8643, Y 18.1870, Z -4.6667, A 0.000, B 0.000, C 0.000 }
gfCNCPoint3[29479] = {X 330.4023, Y 17.4521, Z -4.6667, A 0.000, B 0.000, C 0.000 }
gfCNCPoint3[29480] = {X 326.8820, Y 10.2103, Z -4.6667, A 0.000, B 0.000, C 0.000 }
gfCNCPoint3[29481] = {X 326.5719, Y 9.3163, Z -4.6667, A 0.000, B 0.000, C 0.000 }
gfCNCPoint3[29482] = {X 326.4804, Y 8.3746, Z -4.6667, A 0.000, B 0.000, C 0.000 }
gfCNCPoint3[29483] = {X 326.6127, Y 7.4376, Z -4.6667, A 0.000, B 0.000, C 0.000 }
gfCNCPoint3[29484] = {X 326.9614, Y 6.5580, Z -4.6667, A 0.000, B 0.000, C 0.000 }
gfCNCPoint3[29485] = {X 327.5070, Y 5.7849, Z -4.6667, A 0.000, B 0.000, C 0.000 }
gfCNCPoint3[29486] = {X 328.2189, Y 5.1616, Z -4.6667, A 0.000, B 0.000, C 0.000 }
gfCNCPoint3[29487] = {X 328.8880, Y 4.7034, Z -4.6667, A 0.000, B 0.000, C 0.000 }
gfCNCPoint3[29488] = {X 329.7043, Y 4.2813, Z -4.6667, A 0.000, B 0.000, C 0.000 }
gfCNCPoint3[29489] = {X 330.5954, Y 4.0567, Z -4.6667, A 0.000, B 0.000, C 0.000 }
gfCNCPoint3[29490] = {X 331.5142, Y 4.0413, Z -4.6667, A 0.000, B 0.000, C 0.000 }
gfCNCPoint3[29491] = {X 332.4122, Y 4.2361, Z -4.6667, A 0.000, B 0.000, C 0.000 }
gfCNCPoint3[29492] = {X 332.5467, Y 4.2821, Z -4.6667, A 0.000, B 0.000, C 0.000 }
gfCNCPoint3[29493] = {X 332.6257, Y 4.2345, Z -4.6667, A 0.000, B 0.000, C 0.000 }
gfCNCPoint3[29494] = {X 332.7048, Y 4.1871, Z -4.6667, A 0.000, B 0.000, C 0.000 }
gfCNCPoint3[29495] = {X 334.1611, Y 3.3763, Z -4.6667, A 0.000, B 0.000, C 0.000 }
gfCNCPoint3[29496] = {X 335.6629, Y 2.6534, Z -4.6667, A 0.000, B 0.000, C 0.000 }
gfCNCPoint3[29497] = {X 336.0092, Y 2.4992, Z -4.6667, A 0.000, B 0.000, C 0.000 }
gfCNCPoint3[29498] = {X 338.0805, Y 1.6912, Z -4.6667, A 0.000, B 0.000, C 0.000 }
gfCNCPoint3[29499] = {X 340.2133, Y 1.0633, Z -4.6667, A 0.000, B 0.000, C 0.000 }
gfCNCPoint3[29500] = {X 342.3920, Y 0.6202, Z -4.6667, A 0.000, B 0.000, C 0.000 }
gfCNCPoint3[29501] = {X 344.6007, Y 0.3651, Z -4.6667, A 0.000, B 0.000, C 0.000 }
gfCNCPoint3[29502] = {X 346.8231, Y 0.3000, Z -4.6667, A 0.000, B 0.000, C 0.000 }
gfCNCPoint3[29503] = {X 349.0429, Y 0.4253, Z -4.6667, A 0.000, B 0.000, C 0.000 }
gfCNCPoint3[29504] = {X 351.2438, Y 0.7400, Z -4.6667, A 0.000, B 0.000, C 0.000 }
gfCNCPoint3[29505] = {X 351.5277, Y 0.7930, Z -4.6667, A 0.000, B 0.000, C 0.000 }
gfCNCPoint3[29506] = {X 352.2755, Y -3.2179, Z -4.6667, A 0.000, B 0.000, C 0.000 }
gfCNCPoint3[29507] = {X 352.2755, Y -3.2179, Z -1.6667, A 0.000, B 0.000, C 0.000 }
gfCNCPoint3[29508] = {X 352.2755, Y -3.2179, Z 11.0000, A 0.000, B 0.000, C 0.000 }
gfCNCPoint3[29509] = {X 606.0427, Y 42.9008, Z 11.0000, A 0.000, B 0.000, C 0.000 }
gfCNCPoint3[29510] = {X 606.0427, Y 42.9008, Z -1.6667, A 0.000, B 0.000, C 0.000 }
gfCNCPoint3[29511] = {X 606.0427, Y 42.9008, Z -4.6667, A 0.000, B 0.000, C 0.000 }
gfCNCPoint3[29512] = {X 603.6966, Y 47.0768, Z -4.6667, A 0.000, B 0.000, C 0.000 }
gfCNCPoint3[29513] = {X 603.6311, Y 47.1893, Z -4.6667, A 0.000, B 0.000, C 0.000 }
gfCNCPoint3[29514] = {X 603.5622, Y 47.2997, Z -4.6667, A 0.000, B 0.000, C 0.000 }
gfCNCPoint3[29515] = {X 603.0357, Y 47.9601, Z -4.6667, A 0.000, B 0.000, C 0.000 }
gfCNCPoint3[29516] = {X 602.3889, Y 48.5030, Z -4.6667, A 0.000, B 0.000, C 0.000 }
gfCNCPoint3[29517] = {X 601.6473, Y 48.9069, Z -4.6667, A 0.000, B 0.000, C 0.000 }
gfCNCPoint3[29518] = {X 600.8403, Y 49.1559, Z -4.6667, A 0.000, B 0.000, C 0.000 }
gfCNCPoint3[29519] = {X 600.0000, Y 49.2400, Z -4.6667, A 0.000, B 0.000, C 0.000 }
gfCNCPoint3[29520] = {X 593.5565, Y 49.2400, Z -4.6667, A 0.000, B 0.000, C 0.000 }
gfCNCPoint3[29521] = {X 592.6130, Y 49.1337, Z -4.6667, A 0.000, B 0.000, C 0.000 }
gfCNCPoint3[29522] = {X 591.7169, Y 48.8201, Z -4.6667, A 0.000, B 0.000, C 0.000 }
gfCNCPoint3[29523] = {X 590.9129, Y 48.3150, Z -4.6667, A 0.000, B 0.000, C 0.000 }
gfCNCPoint3[29524] = {X 590.2416, Y 47.6436, Z -4.6667, A 0.000, B 0.000, C 0.000 }
gfCNCPoint3[29525] = {X 589.7364, Y 46.8397, Z -4.6667, A 0.000, B 0.000, C 0.000 }
gfCNCPoint3[29526] = {X 589.4228, Y 45.9435, Z -4.6667, A 0.000, B 0.000, C 0.000 }
gfCNCPoint3[29527] = {X 589.3165, Y 45.0000, Z -4.6667, A 0.000, B 0.000, C 0.000 }
gfCNCPoint3[29528] = {X 589.3165, Y 44.0649, Z -4.6667, A 0.000, B 0.000, C 0.000 }
gfCNCPoint3[29529] = {X 589.4209, Y 43.1447, Z -4.6667, A 0.000, B 0.000, C 0.000 }
gfCNCPoint3[29530] = {X 589.7207, Y 42.2686, Z -4.6667, A 0.000, B 0.000, C 0.000 }
gfCNCPoint3[29531] = {X 590.2020, Y 41.4774, Z -4.6667, A 0.000, B 0.000, C 0.000 }
gfCNCPoint3[29532] = {X 590.8422, Y 40.8082, Z -4.6667, A 0.000, B 0.000, C 0.000 }
gfCNCPoint3[29533] = {X 590.8428, Y 33.1206, Z -4.6667, A 0.000, B 0.000, C 0.000 }
gfCNCPoint3[29534] = {X 585.3714, Y 46.6218, Z -4.6667, A 0.000, B 0.000, C 0.000 }
gfCNCPoint3[29535] = {X 585.0085, Y 47.3114, Z -4.6667, A 0.000, B 0.000, C 0.000 }
gfCNCPoint3[29536] = {X 584.5255, Y 47.9228, Z -4.6667, A 0.000, B 0.000, C 0.000 }
gfCNCPoint3[29537] = {X 583.9387, Y 48.4356, Z -4.6667, A 0.000, B 0.000, C 0.000 }
gfCNCPoint3[29538] = {X 583.2680, Y 48.8323, Z -4.6667, A 0.000, B 0.000, C 0.000 }
gfCNCPoint3[29539] = {X 582.3418, Y 49.1460, Z -4.6667, A 0.000, B 0.000, C 0.000 }
gfCNCPoint3[29540] = {X 581.3682, Y 49.2391, Z -4.6667, A 0.000, B 0.000, C 0.000 }
gfCNCPoint3[29541] = {X 580.3993, Y 49.1068, Z -4.6667, A 0.000, B 0.000, C 0.000 }
gfCNCPoint3[29542] = {X 579.4864, Y 48.7559, Z -4.6667, A 0.000, B 0.000, C 0.000 }
gfCNCPoint3[29543] = {X 578.6782, Y 48.2052, Z -4.6667, A 0.000, B 0.000, C 0.000 }
gfCNCPoint3[29544] = {X 578.0177, Y 47.4840, Z -4.6667, A 0.000, B 0.000, C 0.000 }
gfCNCPoint3[29545] = {X 577.5400, Y 46.6307, Z -4.6667, A 0.000, B 0.000, C 0.000 }
gfCNCPoint3[29546] = {X 571.9389, Y 32.9345, Z -4.6667, A 0.000, B 0.000, C 0.000 }
gfCNCPoint3[29547] = {X 571.9392, Y 40.8084, Z -4.6667, A 0.000, B 0.000, C 0.000 }
gfCNCPoint3[29548] = {X 572.5770, Y 41.4686, Z -4.6667, A 0.000, B 0.000, C 0.000 }
gfCNCPoint3[29549] = {X 573.0577, Y 42.2506, Z -4.6667, A 0.000, B 0.000, C 0.000 }
gfCNCPoint3[29550] = {X 573.3588, Y 43.1178, Z -4.6667, A 0.000, B 0.000, C 0.000 }
gfCNCPoint3[29551] = {X 573.4663, Y 44.0294, Z -4.6667, A 0.000, B 0.000, C 0.000 }
gfCNCPoint3[29552] = {X 573.4664, Y 45.0000, Z -4.6667, A 0.000, B 0.000, C 0.000 }
gfCNCPoint3[29553] = {X 573.3601, Y 45.9435, Z -4.6667, A 0.000, B 0.000, C 0.000 }
gfCNCPoint3[29554] = {X 573.0465, Y 46.8397, Z -4.6667, A 0.000, B 0.000, C 0.000 }
gfCNCPoint3[29555] = {X 572.5414, Y 47.6436, Z -4.6667, A 0.000, B 0.000, C 0.000 }
gfCNCPoint3[29556] = {X 571.8700, Y 48.3150, Z -4.6667, A 0.000, B 0.000, C 0.000 }
gfCNCPoint3[29557] = {X 571.0661, Y 48.8201, Z -4.6667, A 0.000, B 0.000, C 0.000 }
gfCNCPoint3[29558] = {X 570.1699, Y 49.1337, Z -4.6667, A 0.000, B 0.000, C 0.000 }
gfCNCPoint3[29559] = {X 569.2264, Y 49.2400, Z -4.6667, A 0.000, B 0.000, C 0.000 }
gfCNCPoint3[29560] = {X 562.4443, Y 49.2400, Z -4.6667, A 0.000, B 0.000, C 0.000 }
gfCNCPoint3[29561] = {X 561.5008, Y 49.1337, Z -4.6667, A 0.000, B 0.000, C 0.000 }
gfCNCPoint3[29562] = {X 560.6046, Y 48.8201, Z -4.6667, A 0.000, B 0.000, C 0.000 }
gfCNCPoint3[29563] = {X 559.8007, Y 48.3150, Z -4.6667, A 0.000, B 0.000, C 0.000 }
gfCNCPoint3[29564] = {X 559.1293, Y 47.6436, Z -4.6667, A 0.000, B 0.000, C 0.000 }
gfCNCPoint3[29565] = {X 558.6242, Y 46.8397, Z -4.6667, A 0.000, B 0.000, C 0.000 }
gfCNCPoint3[29566] = {X 558.3106, Y 45.9435, Z -4.6667, A 0.000, B 0.000, C 0.000 }
gfCNCPoint3[29567] = {X 558.2043, Y 45.0000, Z -4.6667, A 0.000, B 0.000, C 0.000 }
gfCNCPoint3[29568] = {X 558.2043, Y 44.0650, Z -4.6667, A 0.000, B 0.000, C 0.000 }
gfCNCPoint3[29569] = {X 558.3085, Y 43.1444, Z -4.6667, A 0.000, B 0.000, C 0.000 }
gfCNCPoint3[29570] = {X 558.6086, Y 42.2679, Z -4.6667, A 0.000, B 0.000, C 0.000 }
gfCNCPoint3[29571] = {X 559.0906, Y 41.4767, Z -4.6667, A 0.000, B 0.000, C 0.000 }
gfCNCPoint3[29572] = {X 559.7318, Y 40.8080, Z -4.6667, A 0.000, B 0.000, C 0.000 }
gfCNCPoint3[29573] = {X 559.7318, Y 9.1929, Z -4.6667, A 0.000, B 0.000, C 0.000 }
gfCNCPoint3[29574] = {X 559.0938, Y 8.5325, Z -4.6667, A 0.000, B 0.000, C 0.000 }
gfCNCPoint3[29575] = {X 558.6130, Y 7.7503, Z -4.6667, A 0.000, B 0.000, C 0.000 }
gfCNCPoint3[29576] = {X 558.3118, Y 6.8830, Z -4.6667, A 0.000, B 0.000, C 0.000 }
gfCNCPoint3[29577] = {X 558.2045, Y 5.9711, Z -4.6667, A 0.000, B 0.000, C 0.000 }
gfCNCPoint3[29578] = {X 558.2043, Y 5.0000, Z -4.6667, A 0.000, B 0.000, C 0.000 }
gfCNCPoint3[29579] = {X 558.3106, Y 4.0565, Z -4.6667, A 0.000, B 0.000, C 0.000 }
gfCNCPoint3[29580] = {X 558.6242, Y 3.1603, Z -4.6667, A 0.000, B 0.000, C 0.000 }
gfCNCPoint3[29581] = {X 559.1293, Y 2.3564, Z -4.6667, A 0.000, B 0.000, C 0.000 }
gfCNCPoint3[29582] = {X 559.8007, Y 1.6850, Z -4.6667, A 0.000, B 0.000, C 0.000 }
gfCNCPoint3[29583] = {X 560.6046, Y 1.1799, Z -4.6667, A 0.000, B 0.000, C 0.000 }
gfCNCPoint3[29584] = {X 561.5008, Y 0.8663, Z -4.6667, A 0.000, B 0.000, C 0.000 }
gfCNCPoint3[29585] = {X 562.4443, Y 0.7600, Z -4.6667, A 0.000, B 0.000, C 0.000 }
gfCNCPoint3[29586] = {X 570.9376, Y 0.7600, Z -4.6667, A 0.000, B 0.000, C 0.000 }
gfCNCPoint3[29587] = {X 571.8810, Y 0.8663, Z -4.6667, A 0.000, B 0.000, C 0.000 }
gfCNCPoint3[29588] = {X 572.7772, Y 1.1799, Z -4.6667, A 0.000, B 0.000, C 0.000 }
gfCNCPoint3[29589] = {X 573.5812, Y 1.6850, Z -4.6667, A 0.000, B 0.000, C 0.000 }
gfCNCPoint3[29590] = {X 574.2525, Y 2.3564, Z -4.6667, A 0.000, B 0.000, C 0.000 }
gfCNCPoint3[29591] = {X 574.7577, Y 3.1603, Z -4.6667, A 0.000, B 0.000, C 0.000 }
gfCNCPoint3[29592] = {X 575.0712, Y 4.0565, Z -4.6667, A 0.000, B 0.000, C 0.000 }
gfCNCPoint3[29593] = {X 575.1776, Y 5.0000, Z -4.6667, A 0.000, B 0.000, C 0.000 }
gfCNCPoint3[29594] = {X 575.1776, Y 5.9342, Z -4.6667, A 0.000, B 0.000, C 0.000 }
gfCNCPoint3[29595] = {X 575.1024, Y 6.7291, Z -4.6667, A 0.000, B 0.000, C 0.000 }
gfCNCPoint3[29596] = {X 574.8795, Y 7.4958, Z -4.6667, A 0.000, B 0.000, C 0.000 }
gfCNCPoint3[29597] = {X 574.5168, Y 8.2071, Z -4.6667, A 0.000, B 0.000, C 0.000 }
gfCNCPoint3[29598] = {X 581.1908, Y 24.5815, Z -4.6667, A 0.000, B 0.000, C 0.000 }
gfCNCPoint3[29599] = {X 587.9347, Y 8.0879, Z -4.6667, A 0.000, B 0.000, C 0.000 }
gfCNCPoint3[29600] = {X 587.6158, Y 7.4199, Z -4.6667, A 0.000, B 0.000, C 0.000 }
gfCNCPoint3[29601] = {X 587.4179, Y 6.7066, Z -4.6667, A 0.000, B 0.000, C 0.000 }
gfCNCPoint3[29602] = {X 587.3471, Y 5.9698, Z -4.6667, A 0.000, B 0.000, C 0.000 }
gfCNCPoint3[29603] = {X 587.3470, Y 5.0000, Z -4.6667, A 0.000, B 0.000, C 0.000 }
gfCNCPoint3[29604] = {X 587.4533, Y 4.0565, Z -4.6667, A 0.000, B 0.000, C 0.000 }
gfCNCPoint3[29605] = {X 587.7668, Y 3.1603, Z -4.6667, A 0.000, B 0.000, C 0.000 }
gfCNCPoint3[29606] = {X 588.2720, Y 2.3564, Z -4.6667, A 0.000, B 0.000, C 0.000 }
gfCNCPoint3[29607] = {X 588.9434, Y 1.6850, Z -4.6667, A 0.000, B 0.000, C 0.000 }
gfCNCPoint3[29608] = {X 589.7473, Y 1.1799, Z -4.6667, A 0.000, B 0.000, C 0.000 }
gfCNCPoint3[29609] = {X 590.6435, Y 0.8663, Z -4.6667, A 0.000, B 0.000, C 0.000 }
gfCNCPoint3[29610] = {X 591.5870, Y 0.7600, Z -4.6667, A 0.000, B 0.000, C 0.000 }
gfCNCPoint3[29611] = {X 600.0000, Y 0.7600, Z -4.6667, A 0.000, B 0.000, C 0.000 }
gfCNCPoint3[29612] = {X 600.8403, Y 0.8441, Z -4.6667, A 0.000, B 0.000, C 0.000 }
gfCNCPoint3[29613] = {X 601.6473, Y 1.0931, Z -4.6667, A 0.000, B 0.000, C 0.000 }
gfCNCPoint3[29614] = {X 602.3889, Y 1.4970, Z -4.6667, A 0.000, B 0.000, C 0.000 }
gfCNCPoint3[29615] = {X 603.0357, Y 2.0399, Z -4.6667, A 0.000, B 0.000, C 0.000 }
gfCNCPoint3[29616] = {X 603.5622, Y 2.7003, Z -4.6667, A 0.000, B 0.000, C 0.000 }
gfCNCPoint3[29617] = {X 603.6311, Y 2.8107, Z -4.6667, A 0.000, B 0.000, C 0.000 }
gfCNCPoint3[29618] = {X 603.6966, Y 2.9232, Z -4.6667, A 0.000, B 0.000, C 0.000 }
gfCNCPoint3[29619] = {X 607.8230, Y 10.2681, Z -4.6667, A 0.000, B 0.000, C 0.000 }
gfCNCPoint3[29620] = {X 607.8230, Y 10.2681, Z -1.6667, A 0.000, B 0.000, C 0.000 }
gfCNCPoint3[29621] = {X 607.8230, Y 10.2681, Z 11.0000, A 0.000, B 0.000, C 0.000 }
gfCNCPoint3[29622] = {X 607.6966, Y 39.1590, Z 11.0000, A 0.000, B 0.000, C 0.000 }
gfCNCPoint3[29623] = {X 607.6966, Y 39.1590, Z -1.6667, A 0.000, B 0.000, C 0.000 }
gfCNCPoint3[29624] = {X 607.6966, Y 39.1590, Z -4.6667, A 0.000, B 0.000, C 0.000 }
gfCNCPoint3[29625] = {X 603.6966, Y 46.9081, Z -4.6667, A 0.000, B 0.000, C 0.000 }
gfCNCPoint3[29626] = {X 603.6000, Y 47.0847, Z -4.6667, A 0.000, B 0.000, C 0.000 }
gfCNCPoint3[29627] = {X 603.4949, Y 47.2563, Z -4.6667, A 0.000, B 0.000, C 0.000 }
gfCNCPoint3[29628] = {X 602.9785, Y 47.9042, Z -4.6667, A 0.000, B 0.000, C 0.000 }
gfCNCPoint3[29629] = {X 602.3438, Y 48.4369, Z -4.6667, A 0.000, B 0.000, C 0.000 }
gfCNCPoint3[29630] = {X 601.6162, Y 48.8332, Z -4.6667, A 0.000, B 0.000, C 0.000 }
gfCNCPoint3[29631] = {X 600.8244, Y 49.0775, Z -4.6667, A 0.000, B 0.000, C 0.000 }
gfCNCPoint3[29632] = {X 600.0000, Y 49.1600, Z -4.6667, A 0.000, B 0.000, C 0.000 }
gfCNCPoint3[29633] = {X 593.5565, Y 49.1600, Z -4.6667, A 0.000, B 0.000, C 0.000 }
gfCNCPoint3[29634] = {X 592.6308, Y 49.0557, Z -4.6667, A 0.000, B 0.000, C 0.000 }
gfCNCPoint3[29635] = {X 591.7516, Y 48.7480, Z -4.6667, A 0.000, B 0.000, C 0.000 }
gfCNCPoint3[29636] = {X 590.9628, Y 48.2524, Z -4.6667, A 0.000, B 0.000, C 0.000 }
gfCNCPoint3[29637] = {X 590.3041, Y 47.5937, Z -4.6667, A 0.000, B 0.000, C 0.000 }
gfCNCPoint3[29638] = {X 589.8085, Y 46.8050, Z -4.6667, A 0.000, B 0.000, C 0.000 }
gfCNCPoint3[29639] = {X 589.5008, Y 45.9257, Z -4.6667, A 0.000, B 0.000, C 0.000 }
gfCNCPoint3[29640] = {X 589.3965, Y 45.0000, Z -4.6667, A 0.000, B 0.000, C 0.000 }
gfCNCPoint3[29641] = {X 589.3965, Y 44.0653, Z -4.6667, A 0.000, B 0.000, C 0.000 }
gfCNCPoint3[29642] = {X 589.5010, Y 43.1533, Z -4.6667, A 0.000, B 0.000, C 0.000 }
gfCNCPoint3[29643] = {X 589.8011, Y 42.2857, Z -4.6667, A 0.000, B 0.000, C 0.000 }
gfCNCPoint3[29644] = {X 590.2825, Y 41.5041, Z -4.6667, A 0.000, B 0.000, C 0.000 }
gfCNCPoint3[29645] = {X 590.9222, Y 40.8457, Z -4.6667, A 0.000, B 0.000, C 0.000 }
gfCNCPoint3[29646] = {X 590.9228, Y 32.7101, Z -4.6667, A 0.000, B 0.000, C 0.000 }
gfCNCPoint3[29647] = {X 585.2975, Y 46.5912, Z -4.6667, A 0.000, B 0.000, C 0.000 }
gfCNCPoint3[29648] = {X 584.9414, Y 47.2678, Z -4.6667, A 0.000, B 0.000, C 0.000 }
gfCNCPoint3[29649] = {X 584.4675, Y 47.8677, Z -4.6667, A 0.000, B 0.000, C 0.000 }
gfCNCPoint3[29650] = {X 583.8918, Y 48.3708, Z -4.6667, A 0.000, B 0.000, C 0.000 }
gfCNCPoint3[29651] = {X 583.2338, Y 48.7600, Z -4.6667, A 0.000, B 0.000, C 0.000 }
gfCNCPoint3[29652] = {X 582.3250, Y 49.0678, Z -4.6667, A 0.000, B 0.000, C 0.000 }
gfCNCPoint3[29653] = {X 581.3699, Y 49.1592, Z -4.6667, A 0.000, B 0.000, C 0.000 }
gfCNCPoint3[29654] = {X 580.4192, Y 49.0293, Z -4.6667, A 0.000, B 0.000, C 0.000 }
gfCNCPoint3[29655] = {X 579.5236, Y 48.6850, Z -4.6667, A 0.000, B 0.000, C 0.000 }
gfCNCPoint3[29656] = {X 578.7306, Y 48.1448, Z -4.6667, A 0.000, B 0.000, C 0.000 }
gfCNCPoint3[29657] = {X 578.0826, Y 47.4372, Z -4.6667, A 0.000, B 0.000, C 0.000 }
gfCNCPoint3[29658] = {X 577.6138, Y 46.5999, Z -4.6667, A 0.000, B 0.000, C 0.000 }
gfCNCPoint3[29659] = {X 571.8589, Y 32.5275, Z -4.6667, A 0.000, B 0.000, C 0.000 }
gfCNCPoint3[29660] = {X 571.8592, Y 40.8461, Z -4.6667, A 0.000, B 0.000, C 0.000 }
gfCNCPoint3[29661] = {X 572.4965, Y 41.4956, Z -4.6667, A 0.000, B 0.000, C 0.000 }
gfCNCPoint3[29662] = {X 572.9773, Y 42.2680, Z -4.6667, A 0.000, B 0.000, C 0.000 }
gfCNCPoint3[29663] = {X 573.2787, Y 43.1266, Z -4.6667, A 0.000, B 0.000, C 0.000 }
gfCNCPoint3[29664] = {X 573.3863, Y 44.0301, Z -4.6667, A 0.000, B 0.000, C 0.000 }
gfCNCPoint3[29665] = {X 573.3864, Y 45.0000, Z -4.6667, A 0.000, B 0.000, C 0.000 }
gfCNCPoint3[29666] = {X 573.2821, Y 45.9257, Z -4.6667, A 0.000, B 0.000, C 0.000 }
gfCNCPoint3[29667] = {X 572.9745, Y 46.8050, Z -4.6667, A 0.000, B 0.000, C 0.000 }
gfCNCPoint3[29668] = {X 572.4788, Y 47.5937, Z -4.6667, A 0.000, B 0.000, C 0.000 }
gfCNCPoint3[29669] = {X 571.8201, Y 48.2524, Z -4.6667, A 0.000, B 0.000, C 0.000 }
gfCNCPoint3[29670] = {X 571.0314, Y 48.7480, Z -4.6667, A 0.000, B 0.000, C 0.000 }
gfCNCPoint3[29671] = {X 570.1521, Y 49.0557, Z -4.6667, A 0.000, B 0.000, C 0.000 }
gfCNCPoint3[29672] = {X 569.2264, Y 49.1600, Z -4.6667, A 0.000, B 0.000, C 0.000 }
gfCNCPoint3[29673] = {X 562.4443, Y 49.1600, Z -4.6667, A 0.000, B 0.000, C 0.000 }
gfCNCPoint3[29674] = {X 561.5186, Y 49.0557, Z -4.6667, A 0.000, B 0.000, C 0.000 }
gfCNCPoint3[29675] = {X 560.6393, Y 48.7480, Z -4.6667, A 0.000, B 0.000, C 0.000 }
gfCNCPoint3[29676] = {X 559.8506, Y 48.2524, Z -4.6667, A 0.000, B 0.000, C 0.000 }
gfCNCPoint3[29677] = {X 559.1919, Y 47.5937, Z -4.6667, A 0.000, B 0.000, C 0.000 }
gfCNCPoint3[29678] = {X 558.6963, Y 46.8050, Z -4.6667, A 0.000, B 0.000, C 0.000 }
gfCNCPoint3[29679] = {X 558.3886, Y 45.9257, Z -4.6667, A 0.000, B 0.000, C 0.000 }
gfCNCPoint3[29680] = {X 558.2843, Y 45.0000, Z -4.6667, A 0.000, B 0.000, C 0.000 }
gfCNCPoint3[29681] = {X 558.2843, Y 44.0653, Z -4.6667, A 0.000, B 0.000, C 0.000 }
gfCNCPoint3[29682] = {X 558.3886, Y 43.1529, Z -4.6667, A 0.000, B 0.000, C 0.000 }
gfCNCPoint3[29683] = {X 558.6890, Y 42.2851, Z -4.6667, A 0.000, B 0.000, C 0.000 }
gfCNCPoint3[29684] = {X 559.1711, Y 41.5035, Z -4.6667, A 0.000, B 0.000, C 0.000 }
gfCNCPoint3[29685] = {X 559.8118, Y 40.8455, Z -4.6667, A 0.000, B 0.000, C 0.000 }
gfCNCPoint3[29686] = {X 559.8118, Y 9.1552, Z -4.6667, A 0.000, B 0.000, C 0.000 }
gfCNCPoint3[29687] = {X 559.1743, Y 8.5056, Z -4.6667, A 0.000, B 0.000, C 0.000 }
gfCNCPoint3[29688] = {X 558.6933, Y 7.7329, Z -4.6667, A 0.000, B 0.000, C 0.000 }
gfCNCPoint3[29689] = {X 558.3919, Y 6.8742, Z -4.6667, A 0.000, B 0.000, C 0.000 }
gfCNCPoint3[29690] = {X 558.2845, Y 5.9704, Z -4.6667, A 0.000, B 0.000, C 0.000 }
gfCNCPoint3[29691] = {X 558.2843, Y 5.0000, Z -4.6667, A 0.000, B 0.000, C 0.000 }
gfCNCPoint3[29692] = {X 558.3886, Y 4.0743, Z -4.6667, A 0.000, B 0.000, C 0.000 }
gfCNCPoint3[29693] = {X 558.6963, Y 3.1950, Z -4.6667, A 0.000, B 0.000, C 0.000 }
gfCNCPoint3[29694] = {X 559.1919, Y 2.4063, Z -4.6667, A 0.000, B 0.000, C 0.000 }
gfCNCPoint3[29695] = {X 559.8506, Y 1.7476, Z -4.6667, A 0.000, B 0.000, C 0.000 }
gfCNCPoint3[29696] = {X 560.6393, Y 1.2520, Z -4.6667, A 0.000, B 0.000, C 0.000 }
gfCNCPoint3[29697] = {X 561.5186, Y 0.9443, Z -4.6667, A 0.000, B 0.000, C 0.000 }
gfCNCPoint3[29698] = {X 562.4443, Y 0.8400, Z -4.6667, A 0.000, B 0.000, C 0.000 }
gfCNCPoint3[29699] = {X 570.9376, Y 0.8400, Z -4.6667, A 0.000, B 0.000, C 0.000 }
gfCNCPoint3[29700] = {X 571.8632, Y 0.9443, Z -4.6667, A 0.000, B 0.000, C 0.000 }
gfCNCPoint3[29701] = {X 572.7425, Y 1.2520, Z -4.6667, A 0.000, B 0.000, C 0.000 }
gfCNCPoint3[29702] = {X 573.5313, Y 1.7476, Z -4.6667, A 0.000, B 0.000, C 0.000 }
gfCNCPoint3[29703] = {X 574.1900, Y 2.4063, Z -4.6667, A 0.000, B 0.000, C 0.000 }
gfCNCPoint3[29704] = {X 574.6856, Y 3.1950, Z -4.6667, A 0.000, B 0.000, C 0.000 }
gfCNCPoint3[29705] = {X 574.9933, Y 4.0743, Z -4.6667, A 0.000, B 0.000, C 0.000 }
gfCNCPoint3[29706] = {X 575.0976, Y 5.0000, Z -4.6667, A 0.000, B 0.000, C 0.000 }
gfCNCPoint3[29707] = {X 575.0976, Y 5.9342, Z -4.6667, A 0.000, B 0.000, C 0.000 }
gfCNCPoint3[29708] = {X 575.0212, Y 6.7276, Z -4.6667, A 0.000, B 0.000, C 0.000 }
gfCNCPoint3[29709] = {X 574.7949, Y 7.4918, Z -4.6667, A 0.000, B 0.000, C 0.000 }
gfCNCPoint3[29710] = {X 574.4271, Y 8.1988, Z -4.6667, A 0.000, B 0.000, C 0.000 }
gfCNCPoint3[29711] = {X 581.1907, Y 24.7932, Z -4.6667, A 0.000, B 0.000, C 0.000 }
gfCNCPoint3[29712] = {X 588.0239, Y 8.0812, Z -4.6667, A 0.000, B 0.000, C 0.000 }
gfCNCPoint3[29713] = {X 587.7001, Y 7.4165, Z -4.6667, A 0.000, B 0.000, C 0.000 }
gfCNCPoint3[29714] = {X 587.4990, Y 6.7050, Z -4.6667, A 0.000, B 0.000, C 0.000 }
gfCNCPoint3[29715] = {X 587.4271, Y 5.9692, Z -4.6667, A 0.000, B 0.000, C 0.000 }
gfCNCPoint3[29716] = {X 587.4270, Y 5.0000, Z -4.6667, A 0.000, B 0.000, C 0.000 }
gfCNCPoint3[29717] = {X 587.5313, Y 4.0743, Z -4.6667, A 0.000, B 0.000, C 0.000 }
gfCNCPoint3[29718] = {X 587.8389, Y 3.1950, Z -4.6667, A 0.000, B 0.000, C 0.000 }
gfCNCPoint3[29719] = {X 588.3345, Y 2.4063, Z -4.6667, A 0.000, B 0.000, C 0.000 }
gfCNCPoint3[29720] = {X 588.9932, Y 1.7476, Z -4.6667, A 0.000, B 0.000, C 0.000 }
gfCNCPoint3[29721] = {X 589.7820, Y 1.2520, Z -4.6667, A 0.000, B 0.000, C 0.000 }
gfCNCPoint3[29722] = {X 590.6613, Y 0.9443, Z -4.6667, A 0.000, B 0.000, C 0.000 }
gfCNCPoint3[29723] = {X 591.5870, Y 0.8400, Z -4.6667, A 0.000, B 0.000, C 0.000 }
gfCNCPoint3[29724] = {X 600.0000, Y 0.8400, Z -4.6667, A 0.000, B 0.000, C 0.000 }
gfCNCPoint3[29725] = {X 600.8244, Y 0.9225, Z -4.6667, A 0.000, B 0.000, C 0.000 }
gfCNCPoint3[29726] = {X 601.6162, Y 1.1668, Z -4.6667, A 0.000, B 0.000, C 0.000 }
gfCNCPoint3[29727] = {X 602.3438, Y 1.5631, Z -4.6667, A 0.000, B 0.000, C 0.000 }
gfCNCPoint3[29728] = {X 602.9785, Y 2.0958, Z -4.6667, A 0.000, B 0.000, C 0.000 }
gfCNCPoint3[29729] = {X 603.4949, Y 2.7437, Z -4.6667, A 0.000, B 0.000, C 0.000 }
gfCNCPoint3[29730] = {X 603.6000, Y 2.9153, Z -4.6667, A 0.000, B 0.000, C 0.000 }
gfCNCPoint3[29731] = {X 603.6966, Y 3.0919, Z -4.6667, A 0.000, B 0.000, C 0.000 }
gfCNCPoint3[29732] = {X 607.6966, Y 10.8410, Z -4.6667, A 0.000, B 0.000, C 0.000 }
gfCNCPoint3[29733] = {X 607.6966, Y 10.8410, Z -1.6667, A 0.000, B 0.000, C 0.000 }
gfCNCPoint3[29734] = {X 607.6966, Y 10.8410, Z 11.0000, A 0.000, B 0.000, C 0.000 }
gfCNCPoint3[29735] = {X 607.6966, Y 38.1638, Z 11.0000, A 0.000, B 0.000, C 0.000 }
gfCNCPoint3[29736] = {X 607.6966, Y 38.1638, Z -1.6667, A 0.000, B 0.000, C 0.000 }
gfCNCPoint3[29737] = {X 607.6966, Y 38.1638, Z -4.6667, A 0.000, B 0.000, C 0.000 }
gfCNCPoint3[29738] = {X 603.6966, Y 46.7268, Z -4.6667, A 0.000, B 0.000, C 0.000 }
gfCNCPoint3[29739] = {X 603.5704, Y 46.9744, Z -4.6667, A 0.000, B 0.000, C 0.000 }
gfCNCPoint3[29740] = {X 603.4277, Y 47.2129, Z -4.6667, A 0.000, B 0.000, C 0.000 }
gfCNCPoint3[29741] = {X 602.9212, Y 47.8484, Z -4.6667, A 0.000, B 0.000, C 0.000 }
gfCNCPoint3[29742] = {X 602.2987, Y 48.3708, Z -4.6667, A 0.000, B 0.000, C 0.000 }
gfCNCPoint3[29743] = {X 601.5851, Y 48.7595, Z -4.6667, A 0.000, B 0.000, C 0.000 }
gfCNCPoint3[29744] = {X 600.8086, Y 48.9991, Z -4.6667, A 0.000, B 0.000, C 0.000 }
gfCNCPoint3[29745] = {X 600.0000, Y 49.0800, Z -4.6667, A 0.000, B 0.000, C 0.000 }
gfCNCPoint3[29746] = {X 593.5565, Y 49.0800, Z -4.6667, A 0.000, B 0.000, C 0.000 }
gfCNCPoint3[29747] = {X 592.6486, Y 48.9777, Z -4.6667, A 0.000, B 0.000, C 0.000 }
gfCNCPoint3[29748] = {X 591.7863, Y 48.6760, Z -4.6667, A 0.000, B 0.000, C 0.000 }
gfCNCPoint3[29749] = {X 591.0127, Y 48.1899, Z -4.6667, A 0.000, B 0.000, C 0.000 }
gfCNCPoint3[29750] = {X 590.3667, Y 47.5438, Z -4.6667, A 0.000, B 0.000, C 0.000 }
gfCNCPoint3[29751] = {X 589.8806, Y 46.7702, Z -4.6667, A 0.000, B 0.000, C 0.000 }
gfCNCPoint3[29752] = {X 589.5788, Y 45.9079, Z -4.6667, A 0.000, B 0.000, C 0.000 }
gfCNCPoint3[29753] = {X 589.4765, Y 45.0000, Z -4.6667, A 0.000, B 0.000, C 0.000 }
gfCNCPoint3[29754] = {X 589.4765, Y 44.0656, Z -4.6667, A 0.000, B 0.000, C 0.000 }
gfCNCPoint3[29755] = {X 589.5811, Y 43.1618, Z -4.6667, A 0.000, B 0.000, C 0.000 }
gfCNCPoint3[29756] = {X 589.8815, Y 42.3030, Z -4.6667, A 0.000, B 0.000, C 0.000 }
gfCNCPoint3[29757] = {X 590.3630, Y 41.5311, Z -4.6667, A 0.000, B 0.000, C 0.000 }
gfCNCPoint3[29758] = {X 591.0022, Y 40.8836, Z -4.6667, A 0.000, B 0.000, C 0.000 }
gfCNCPoint3[29759] = {X 591.0028, Y 32.2996, Z -4.6667, A 0.000, B 0.000, C 0.000 }
gfCNCPoint3[29760] = {X 585.2236, Y 46.5606, Z -4.6667, A 0.000, B 0.000, C 0.000 }
gfCNCPoint3[29761] = {X 584.8743, Y 47.2242, Z -4.6667, A 0.000, B 0.000, C 0.000 }
gfCNCPoint3[29762] = {X 584.4095, Y 47.8125, Z -4.6667, A 0.000, B 0.000, C 0.000 }
gfCNCPoint3[29763] = {X 583.8449, Y 48.3059, Z -4.6667, A 0.000, B 0.000, C 0.000 }
gfCNCPoint3[29764] = {X 583.1996, Y 48.6877, Z -4.6667, A 0.000, B 0.000, C 0.000 }
gfCNCPoint3[29765] = {X 582.3082, Y 48.9895, Z -4.6667, A 0.000, B 0.000, C 0.000 }
gfCNCPoint3[29766] = {X 581.3715, Y 49.0792, Z -4.6667, A 0.000, B 0.000, C 0.000 }
gfCNCPoint3[29767] = {X 580.4391, Y 48.9518, Z -4.6667, A 0.000, B 0.000, C 0.000 }
gfCNCPoint3[29768] = {X 579.5607, Y 48.6142, Z -4.6667, A 0.000, B 0.000, C 0.000 }
gfCNCPoint3[29769] = {X 578.7830, Y 48.0843, Z -4.6667, A 0.000, B 0.000, C 0.000 }
gfCNCPoint3[29770] = {X 578.1474, Y 47.3903, Z -4.6667, A 0.000, B 0.000, C 0.000 }
gfCNCPoint3[29771] = {X 577.6877, Y 46.5692, Z -4.6667, A 0.000, B 0.000, C 0.000 }
gfCNCPoint3[29772] = {X 571.7789, Y 32.1205, Z -4.6667, A 0.000, B 0.000, C 0.000 }
gfCNCPoint3[29773] = {X 571.7792, Y 40.8841, Z -4.6667, A 0.000, B 0.000, C 0.000 }
gfCNCPoint3[29774] = {X 571.8685, Y 40.9569, Z -4.6667, A 0.000, B 0.000, C 0.000 }
gfCNCPoint3[29775] = {X 572.4696, Y 41.5904, Z -4.6667, A 0.000, B 0.000, C 0.000 }
gfCNCPoint3[29776] = {X 572.9221, Y 42.3373, Z -4.6667, A 0.000, B 0.000, C 0.000 }
gfCNCPoint3[29777] = {X 573.2053, Y 43.1634, Z -4.6667, A 0.000, B 0.000, C 0.000 }
gfCNCPoint3[29778] = {X 573.3063, Y 44.0308, Z -4.6667, A 0.000, B 0.000, C 0.000 }
gfCNCPoint3[29779] = {X 573.3064, Y 45.0000, Z -4.6667, A 0.000, B 0.000, C 0.000 }
gfCNCPoint3[29780] = {X 573.2041, Y 45.9079, Z -4.6667, A 0.000, B 0.000, C 0.000 }
gfCNCPoint3[29781] = {X 572.9024, Y 46.7702, Z -4.6667, A 0.000, B 0.000, C 0.000 }
gfCNCPoint3[29782] = {X 572.4163, Y 47.5438, Z -4.6667, A 0.000, B 0.000, C 0.000 }
gfCNCPoint3[29783] = {X 571.7703, Y 48.1899, Z -4.6667, A 0.000, B 0.000, C 0.000 }
gfCNCPoint3[29784] = {X 570.9967, Y 48.6760, Z -4.6667, A 0.000, B 0.000, C 0.000 }
gfCNCPoint3[29785] = {X 570.1343, Y 48.9777, Z -4.6667, A 0.000, B 0.000, C 0.000 }
gfCNCPoint3[29786] = {X 569.2264, Y 49.0800, Z -4.6667, A 0.000, B 0.000, C 0.000 }
gfCNCPoint3[29787] = {X 562.4443, Y 49.0800, Z -4.6667, A 0.000, B 0.000, C 0.000 }
gfCNCPoint3[29788] = {X 561.5364, Y 48.9777, Z -4.6667, A 0.000, B 0.000, C 0.000 }
gfCNCPoint3[29789] = {X 560.6741, Y 48.6760, Z -4.6667, A 0.000, B 0.000, C 0.000 }
gfCNCPoint3[29790] = {X 559.9005, Y 48.1899, Z -4.6667, A 0.000, B 0.000, C 0.000 }
gfCNCPoint3[29791] = {X 559.2544, Y 47.5438, Z -4.6667, A 0.000, B 0.000, C 0.000 }
gfCNCPoint3[29792] = {X 558.7683, Y 46.7702, Z -4.6667, A 0.000, B 0.000, C 0.000 }
gfCNCPoint3[29793] = {X 558.4666, Y 45.9079, Z -4.6667, A 0.000, B 0.000, C 0.000 }
gfCNCPoint3[29794] = {X 558.3643, Y 45.0000, Z -4.6667, A 0.000, B 0.000, C 0.000 }
gfCNCPoint3[29795] = {X 558.3643, Y 44.0657, Z -4.6667, A 0.000, B 0.000, C 0.000 }
gfCNCPoint3[29796] = {X 558.4608, Y 43.1966, Z -4.6667, A 0.000, B 0.000, C 0.000 }
gfCNCPoint3[29797] = {X 558.7388, Y 42.3675, Z -4.6667, A 0.000, B 0.000, C 0.000 }
gfCNCPoint3[29798] = {X 559.1858, Y 41.6160, Z -4.6667, A 0.000, B 0.000, C 0.000 }
gfCNCPoint3[29799] = {X 559.7815, Y 40.9759, Z -4.6667, A 0.000, B 0.000, C 0.000 }
gfCNCPoint3[29800] = {X 559.8363, Y 40.9292, Z -4.6667, A 0.000, B 0.000, C 0.000 }
gfCNCPoint3[29801] = {X 559.8918, Y 40.8835, Z -4.6667, A 0.000, B 0.000, C 0.000 }
gfCNCPoint3[29802] = {X 559.8918, Y 9.1170, Z -4.6667, A 0.000, B 0.000, C 0.000 }
gfCNCPoint3[29803] = {X 559.8358, Y 9.0713, Z -4.6667, A 0.000, B 0.000, C 0.000 }
gfCNCPoint3[29804] = {X 559.7807, Y 9.0246, Z -4.6667, A 0.000, B 0.000, C 0.000 }
gfCNCPoint3[29805] = {X 559.1883, Y 8.3928, Z -4.6667, A 0.000, B 0.000, C 0.000 }
gfCNCPoint3[29806] = {X 558.7427, Y 7.6501, Z -4.6667, A 0.000, B 0.000, C 0.000 }
gfCNCPoint3[29807] = {X 558.4639, Y 6.8301, Z -4.6667, A 0.000, B 0.000, C 0.000 }
gfCNCPoint3[29808] = {X 558.3645, Y 5.9697, Z -4.6667, A 0.000, B 0.000, C 0.000 }
gfCNCPoint3[29809] = {X 558.3643, Y 5.0000, Z -4.6667, A 0.000, B 0.000, C 0.000 }
gfCNCPoint3[29810] = {X 558.4666, Y 4.0921, Z -4.6667, A 0.000, B 0.000, C 0.000 }
gfCNCPoint3[29811] = {X 558.7683, Y 3.2298, Z -4.6667, A 0.000, B 0.000, C 0.000 }
gfCNCPoint3[29812] = {X 559.2544, Y 2.4562, Z -4.6667, A 0.000, B 0.000, C 0.000 }
gfCNCPoint3[29813] = {X 559.9005, Y 1.8101, Z -4.6667, A 0.000, B 0.000, C 0.000 }
gfCNCPoint3[29814] = {X 560.6741, Y 1.3240, Z -4.6667, A 0.000, B 0.000, C 0.000 }
gfCNCPoint3[29815] = {X 561.5364, Y 1.0223, Z -4.6667, A 0.000, B 0.000, C 0.000 }
gfCNCPoint3[29816] = {X 562.4443, Y 0.9200, Z -4.6667, A 0.000, B 0.000, C 0.000 }
gfCNCPoint3[29817] = {X 570.9376, Y 0.9200, Z -4.6667, A 0.000, B 0.000, C 0.000 }
gfCNCPoint3[29818] = {X 571.8454, Y 1.0223, Z -4.6667, A 0.000, B 0.000, C 0.000 }
gfCNCPoint3[29819] = {X 572.7078, Y 1.3240, Z -4.6667, A 0.000, B 0.000, C 0.000 }
gfCNCPoint3[29820] = {X 573.4814, Y 1.8101, Z -4.6667, A 0.000, B 0.000, C 0.000 }
gfCNCPoint3[29821] = {X 574.1274, Y 2.4562, Z -4.6667, A 0.000, B 0.000, C 0.000 }
gfCNCPoint3[29822] = {X 574.6135, Y 3.2298, Z -4.6667, A 0.000, B 0.000, C 0.000 }
gfCNCPoint3[29823] = {X 574.9153, Y 4.0921, Z -4.6667, A 0.000, B 0.000, C 0.000 }
gfCNCPoint3[29824] = {X 575.0176, Y 5.0000, Z -4.6667, A 0.000, B 0.000, C 0.000 }
gfCNCPoint3[29825] = {X 575.0176, Y 5.9342, Z -4.6667, A 0.000, B 0.000, C 0.000 }
gfCNCPoint3[29826] = {X 574.9500, Y 6.6736, Z -4.6667, A 0.000, B 0.000, C 0.000 }
gfCNCPoint3[29827] = {X 574.7495, Y 7.3884, Z -4.6667, A 0.000, B 0.000, C 0.000 }
gfCNCPoint3[29828] = {X 574.4229, Y 8.0551, Z -4.6667, A 0.000, B 0.000, C 0.000 }
gfCNCPoint3[29829] = {X 574.3785, Y 8.1264, Z -4.6667, A 0.000, B 0.000, C 0.000 }
gfCNCPoint3[29830] = {X 574.3327, Y 8.1967, Z -4.6667, A 0.000, B 0.000, C 0.000 }
gfCNCPoint3[29831] = {X 574.3585, Y 8.2415, Z -4.6667, A 0.000, B 0.000, C 0.000 }
gfCNCPoint3[29832] = {X 581.1906, Y 25.0048, Z -4.6667, A 0.000, B 0.000, C 0.000 }
gfCNCPoint3[29833] = {X 588.1132, Y 8.0741, Z -4.6667, A 0.000, B 0.000, C 0.000 }
gfCNCPoint3[29834] = {X 588.0738, Y 8.0086, Z -4.6667, A 0.000, B 0.000, C 0.000 }
gfCNCPoint3[29835] = {X 588.0355, Y 7.9424, Z -4.6667, A 0.000, B 0.000, C 0.000 }
gfCNCPoint3[29836] = {X 587.7486, Y 7.3175, Z -4.6667, A 0.000, B 0.000, C 0.000 }
gfCNCPoint3[29837] = {X 587.5708, Y 6.6532, Z -4.6667, A 0.000, B 0.000, C 0.000 }
gfCNCPoint3[29838] = {X 587.5071, Y 5.9685, Z -4.6667, A 0.000, B 0.000, C 0.000 }
gfCNCPoint3[29839] = {X 587.5070, Y 5.0000, Z -4.6667, A 0.000, B 0.000, C 0.000 }
gfCNCPoint3[29840] = {X 587.6092, Y 4.0921, Z -4.6667, A 0.000, B 0.000, C 0.000 }
gfCNCPoint3[29841] = {X 587.9110, Y 3.2298, Z -4.6667, A 0.000, B 0.000, C 0.000 }
gfCNCPoint3[29842] = {X 588.3971, Y 2.4562, Z -4.6667, A 0.000, B 0.000, C 0.000 }
gfCNCPoint3[29843] = {X 589.0431, Y 1.8101, Z -4.6667, A 0.000, B 0.000, C 0.000 }
gfCNCPoint3[29844] = {X 589.8167, Y 1.3240, Z -4.6667, A 0.000, B 0.000, C 0.000 }
gfCNCPoint3[29845] = {X 590.6791, Y 1.0223, Z -4.6667, A 0.000, B 0.000, C 0.000 }
gfCNCPoint3[29846] = {X 591.5870, Y 0.9200, Z -4.6667, A 0.000, B 0.000, C 0.000 }
gfCNCPoint3[29847] = {X 600.0000, Y 0.9200, Z -4.6667, A 0.000, B 0.000, C 0.000 }
gfCNCPoint3[29848] = {X 600.8086, Y 1.0009, Z -4.6667, A 0.000, B 0.000, C 0.000 }
gfCNCPoint3[29849] = {X 601.5851, Y 1.2405, Z -4.6667, A 0.000, B 0.000, C 0.000 }
gfCNCPoint3[29850] = {X 602.2987, Y 1.6292, Z -4.6667, A 0.000, B 0.000, C 0.000 }
gfCNCPoint3[29851] = {X 602.9212, Y 2.1516, Z -4.6667, A 0.000, B 0.000, C 0.000 }
gfCNCPoint3[29852] = {X 603.4277, Y 2.7871, Z -4.6667, A 0.000, B 0.000, C 0.000 }
gfCNCPoint3[29853] = {X 603.5704, Y 3.0256, Z -4.6667, A 0.000, B 0.000, C 0.000 }
gfCNCPoint3[29854] = {X 603.6966, Y 3.2732, Z -4.6667, A 0.000, B 0.000, C 0.000 }
gfCNCPoint3[29855] = {X 607.6966, Y 11.8362, Z -4.6667, A 0.000, B 0.000, C 0.000 }
gfCNCPoint3[29856] = {X 607.6966, Y 11.8362, Z -1.6667, A 0.000, B 0.000, C 0.000 }
gfCNCPoint3[29857] = {X 607.6966, Y 11.8362, Z 11.0000, A 0.000, B 0.000, C 0.000 }
gfCNCPoint3[29858] = {X 607.6966, Y 36.8524, Z 11.0000, A 0.000, B 0.000, C 0.000 }
gfCNCPoint3[29859] = {X 607.6966, Y 36.8524, Z -1.6667, A 0.000, B 0.000, C 0.000 }
gfCNCPoint3[29860] = {X 607.6966, Y 36.8524, Z -4.6667, A 0.000, B 0.000, C 0.000 }
gfCNCPoint3[29861] = {X 603.6966, Y 46.5282, Z -4.6667, A 0.000, B 0.000, C 0.000 }
gfCNCPoint3[29862] = {X 603.5431, Y 46.8565, Z -4.6667, A 0.000, B 0.000, C 0.000 }
gfCNCPoint3[29863] = {X 603.3605, Y 47.1695, Z -4.6667, A 0.000, B 0.000, C 0.000 }
gfCNCPoint3[29864] = {X 602.8639, Y 47.7925, Z -4.6667, A 0.000, B 0.000, C 0.000 }
gfCNCPoint3[29865] = {X 602.2537, Y 48.3047, Z -4.6667, A 0.000, B 0.000, C 0.000 }
gfCNCPoint3[29866] = {X 601.5540, Y 48.6858, Z -4.6667, A 0.000, B 0.000, C 0.000 }
gfCNCPoint3[29867] = {X 600.7927, Y 48.9207, Z -4.6667, A 0.000, B 0.000, C 0.000 }
gfCNCPoint3[29868] = {X 600.0000, Y 49.0000, Z -4.6667, A 0.000, B 0.000, C 0.000 }
gfCNCPoint3[29869] = {X 593.5565, Y 49.0000, Z -4.6667, A 0.000, B 0.000, C 0.000 }
gfCNCPoint3[29870] = {X 592.6664, Y 48.8997, Z -4.6667, A 0.000, B 0.000, C 0.000 }
gfCNCPoint3[29871] = {X 591.8210, Y 48.6039, Z -4.6667, A 0.000, B 0.000, C 0.000 }
gfCNCPoint3[29872] = {X 591.0626, Y 48.1273, Z -4.6667, A 0.000, B 0.000, C 0.000 }
gfCNCPoint3[29873] = {X 590.4292, Y 47.4940, Z -4.6667, A 0.000, B 0.000, C 0.000 }
gfCNCPoint3[29874] = {X 589.9527, Y 46.7355, Z -4.6667, A 0.000, B 0.000, C 0.000 }
gfCNCPoint3[29875] = {X 589.6568, Y 45.8901, Z -4.6667, A 0.000, B 0.000, C 0.000 }
gfCNCPoint3[29876] = {X 589.5565, Y 45.0000, Z -4.6667, A 0.000, B 0.000, C 0.000 }
gfCNCPoint3[29877] = {X 589.5565, Y 44.0660, Z -4.6667, A 0.000, B 0.000, C 0.000 }
gfCNCPoint3[29878] = {X 589.6612, Y 43.1705, Z -4.6667, A 0.000, B 0.000, C 0.000 }
gfCNCPoint3[29879] = {X 589.9618, Y 42.3206, Z -4.6667, A 0.000, B 0.000, C 0.000 }
gfCNCPoint3[29880] = {X 590.4434, Y 41.5584, Z -4.6667, A 0.000, B 0.000, C 0.000 }
gfCNCPoint3[29881] = {X 591.0821, Y 40.9221, Z -4.6667, A 0.000, B 0.000, C 0.000 }
gfCNCPoint3[29882] = {X 591.0827, Y 40.7355, Z -4.6667, A 0.000, B 0.000, C 0.000 }
gfCNCPoint3[29883] = {X 591.0841, Y 40.3068, Z -4.6667, A 0.000, B 0.000, C 0.000 }
gfCNCPoint3[29884] = {X 591.0828, Y 32.0433, Z -4.6667, A 0.000, B 0.000, C 0.000 }
gfCNCPoint3[29885] = {X 590.9675, Y 32.1736, Z -4.6667, A 0.000, B 0.000, C 0.000 }
gfCNCPoint3[29886] = {X 590.3124, Y 33.7904, Z -4.6667, A 0.000, B 0.000, C 0.000 }
gfCNCPoint3[29887] = {X 585.1497, Y 46.5300, Z -4.6667, A 0.000, B 0.000, C 0.000 }
gfCNCPoint3[29888] = {X 584.8073, Y 47.1805, Z -4.6667, A 0.000, B 0.000, C 0.000 }
gfCNCPoint3[29889] = {X 584.3516, Y 47.7574, Z -4.6667, A 0.000, B 0.000, C 0.000 }
gfCNCPoint3[29890] = {X 583.7980, Y 48.2411, Z -4.6667, A 0.000, B 0.000, C 0.000 }
gfCNCPoint3[29891] = {X 583.1653, Y 48.6154, Z -4.6667, A 0.000, B 0.000, C 0.000 }
gfCNCPoint3[29892] = {X 582.2878, Y 48.9121, Z -4.6667, A 0.000, B 0.000, C 0.000 }
gfCNCPoint3[29893] = {X 581.3656, Y 48.9990, Z -4.6667, A 0.000, B 0.000, C 0.000 }
gfCNCPoint3[29894] = {X 580.4480, Y 48.8715, Z -4.6667, A 0.000, B 0.000, C 0.000 }
gfCNCPoint3[29895] = {X 579.5845, Y 48.5363, Z -4.6667, A 0.000, B 0.000, C 0.000 }
gfCNCPoint3[29896] = {X 578.8212, Y 48.0115, Z -4.6667, A 0.000, B 0.000, C 0.000 }
gfCNCPoint3[29897] = {X 578.1990, Y 47.3251, Z -4.6667, A 0.000, B 0.000, C 0.000 }
gfCNCPoint3[29898] = {X 577.7515, Y 46.5141, Z -4.6667, A 0.000, B 0.000, C 0.000 }
gfCNCPoint3[29899] = {X 571.6988, Y 31.7135, Z -4.6667, A 0.000, B 0.000, C 0.000 }
gfCNCPoint3[29900] = {X 571.6992, Y 40.9221, Z -4.6667, A 0.000, B 0.000, C 0.000 }
gfCNCPoint3[29901] = {X 571.8380, Y 41.0362, Z -4.6667, A 0.000, B 0.000, C 0.000 }
gfCNCPoint3[29902] = {X 572.4239, Y 41.6626, Z -4.6667, A 0.000, B 0.000, C 0.000 }
gfCNCPoint3[29903] = {X 572.8628, Y 42.3996, Z -4.6667, A 0.000, B 0.000, C 0.000 }
gfCNCPoint3[29904] = {X 573.1345, Y 43.2132, Z -4.6667, A 0.000, B 0.000, C 0.000 }
gfCNCPoint3[29905] = {X 573.2264, Y 44.0660, Z -4.6667, A 0.000, B 0.000, C 0.000 }
gfCNCPoint3[29906] = {X 573.2264, Y 45.0000, Z -4.6667, A 0.000, B 0.000, C 0.000 }
gfCNCPoint3[29907] = {X 573.1261, Y 45.8901, Z -4.6667, A 0.000, B 0.000, C 0.000 }
gfCNCPoint3[29908] = {X 572.8303, Y 46.7355, Z -4.6667, A 0.000, B 0.000, C 0.000 }
gfCNCPoint3[29909] = {X 572.3538, Y 47.4940, Z -4.6667, A 0.000, B 0.000, C 0.000 }
gfCNCPoint3[29910] = {X 571.7204, Y 48.1273, Z -4.6667, A 0.000, B 0.000, C 0.000 }
gfCNCPoint3[29911] = {X 570.9620, Y 48.6039, Z -4.6667, A 0.000, B 0.000, C 0.000 }
gfCNCPoint3[29912] = {X 570.1165, Y 48.8997, Z -4.6667, A 0.000, B 0.000, C 0.000 }
gfCNCPoint3[29913] = {X 569.2264, Y 49.0000, Z -4.6667, A 0.000, B 0.000, C 0.000 }
gfCNCPoint3[29914] = {X 562.4443, Y 49.0000, Z -4.6667, A 0.000, B 0.000, C 0.000 }
gfCNCPoint3[29915] = {X 561.5542, Y 48.8997, Z -4.6667, A 0.000, B 0.000, C 0.000 }
gfCNCPoint3[29916] = {X 560.7088, Y 48.6039, Z -4.6667, A 0.000, B 0.000, C 0.000 }
gfCNCPoint3[29917] = {X 559.9503, Y 48.1273, Z -4.6667, A 0.000, B 0.000, C 0.000 }
gfCNCPoint3[29918] = {X 559.3170, Y 47.4940, Z -4.6667, A 0.000, B 0.000, C 0.000 }
gfCNCPoint3[29919] = {X 558.8404, Y 46.7355, Z -4.6667, A 0.000, B 0.000, C 0.000 }
gfCNCPoint3[29920] = {X 558.5446, Y 45.8901, Z -4.6667, A 0.000, B 0.000, C 0.000 }
gfCNCPoint3[29921] = {X 558.4443, Y 45.0000, Z -4.6667, A 0.000, B 0.000, C 0.000 }
gfCNCPoint3[29922] = {X 558.4443, Y 44.0660, Z -4.6667, A 0.000, B 0.000, C 0.000 }
gfCNCPoint3[29923] = {X 558.5389, Y 43.2138, Z -4.6667, A 0.000, B 0.000, C 0.000 }
gfCNCPoint3[29924] = {X 558.8115, Y 42.4009, Z -4.6667, A 0.000, B 0.000, C 0.000 }
gfCNCPoint3[29925] = {X 559.2498, Y 41.6639, Z -4.6667, A 0.000, B 0.000, C 0.000 }
gfCNCPoint3[29926] = {X 559.8340, Y 41.0363, Z -4.6667, A 0.000, B 0.000, C 0.000 }
gfCNCPoint3[29927] = {X 559.9022, Y 40.9783, Z -4.6667, A 0.000, B 0.000, C 0.000 }
gfCNCPoint3[29928] = {X 559.9718, Y 40.9219, Z -4.6667, A 0.000, B 0.000, C 0.000 }
gfCNCPoint3[29929] = {X 559.9718, Y 9.0784, Z -4.6667, A 0.000, B 0.000, C 0.000 }
gfCNCPoint3[29930] = {X 559.9017, Y 9.0220, Z -4.6667, A 0.000, B 0.000, C 0.000 }
gfCNCPoint3[29931] = {X 559.8329, Y 8.9640, Z -4.6667, A 0.000, B 0.000, C 0.000 }
gfCNCPoint3[29932] = {X 559.2469, Y 8.3375, Z -4.6667, A 0.000, B 0.000, C 0.000 }
gfCNCPoint3[29933] = {X 558.8080, Y 7.6005, Z -4.6667, A 0.000, B 0.000, C 0.000 }
gfCNCPoint3[29934] = {X 558.5363, Y 6.7868, Z -4.6667, A 0.000, B 0.000, C 0.000 }
gfCNCPoint3[29935] = {X 558.4443, Y 5.9340, Z -4.6667, A 0.000, B 0.000, C 0.000 }
gfCNCPoint3[29936] = {X 558.4443, Y 5.0000, Z -4.6667, A 0.000, B 0.000, C 0.000 }
gfCNCPoint3[29937] = {X 558.5446, Y 4.1099, Z -4.6667, A 0.000, B 0.000, C 0.000 }
gfCNCPoint3[29938] = {X 558.8404, Y 3.2645, Z -4.6667, A 0.000, B 0.000, C 0.000 }
gfCNCPoint3[29939] = {X 559.3170, Y 2.5060, Z -4.6667, A 0.000, B 0.000, C 0.000 }
gfCNCPoint3[29940] = {X 559.9503, Y 1.8727, Z -4.6667, A 0.000, B 0.000, C 0.000 }
gfCNCPoint3[29941] = {X 560.7088, Y 1.3961, Z -4.6667, A 0.000, B 0.000, C 0.000 }
gfCNCPoint3[29942] = {X 561.5542, Y 1.1003, Z -4.6667, A 0.000, B 0.000, C 0.000 }
gfCNCPoint3[29943] = {X 562.4443, Y 1.0000, Z -4.6667, A 0.000, B 0.000, C 0.000 }
gfCNCPoint3[29944] = {X 570.9376, Y 1.0000, Z -4.6667, A 0.000, B 0.000, C 0.000 }
gfCNCPoint3[29945] = {X 571.8276, Y 1.1003, Z -4.6667, A 0.000, B 0.000, C 0.000 }
gfCNCPoint3[29946] = {X 572.6731, Y 1.3961, Z -4.6667, A 0.000, B 0.000, C 0.000 }
gfCNCPoint3[29947] = {X 573.4315, Y 1.8727, Z -4.6667, A 0.000, B 0.000, C 0.000 }
gfCNCPoint3[29948] = {X 574.0649, Y 2.5060, Z -4.6667, A 0.000, B 0.000, C 0.000 }
gfCNCPoint3[29949] = {X 574.5414, Y 3.2645, Z -4.6667, A 0.000, B 0.000, C 0.000 }
gfCNCPoint3[29950] = {X 574.8373, Y 4.1099, Z -4.6667, A 0.000, B 0.000, C 0.000 }
gfCNCPoint3[29951] = {X 574.9376, Y 5.0000, Z -4.6667, A 0.000, B 0.000, C 0.000 }
gfCNCPoint3[29952] = {X 574.9372, Y 5.9858, Z -4.6667, A 0.000, B 0.000, C 0.000 }
gfCNCPoint3[29953] = {X 574.8649, Y 6.6929, Z -4.6667, A 0.000, B 0.000, C 0.000 }
gfCNCPoint3[29954] = {X 574.6686, Y 7.3760, Z -4.6667, A 0.000, B 0.000, C 0.000 }
gfCNCPoint3[29955] = {X 574.3545, Y 8.0135, Z -4.6667, A 0.000, B 0.000, C 0.000 }
gfCNCPoint3[29956] = {X 574.2919, Y 8.1131, Z -4.6667, A 0.000, B 0.000, C 0.000 }
gfCNCPoint3[29957] = {X 574.2264, Y 8.2108, Z -4.6667, A 0.000, B 0.000, C 0.000 }
gfCNCPoint3[29958] = {X 574.2611, Y 8.2359, Z -4.6667, A 0.000, B 0.000, C 0.000 }
gfCNCPoint3[29959] = {X 574.2845, Y 8.2719, Z -4.6667, A 0.000, B 0.000, C 0.000 }
gfCNCPoint3[29960] = {X 574.9161, Y 9.8078, Z -4.6667, A 0.000, B 0.000, C 0.000 }
gfCNCPoint3[29961] = {X 581.1904, Y 25.2166, Z -4.6667, A 0.000, B 0.000, C 0.000 }
gfCNCPoint3[29962] = {X 588.2028, Y 8.0665, Z -4.6667, A 0.000, B 0.000, C 0.000 }
gfCNCPoint3[29963] = {X 588.1530, Y 7.9854, Z -4.6667, A 0.000, B 0.000, C 0.000 }
gfCNCPoint3[29964] = {X 588.1051, Y 7.9031, Z -4.6667, A 0.000, B 0.000, C 0.000 }
gfCNCPoint3[29965] = {X 587.8201, Y 7.2797, Z -4.6667, A 0.000, B 0.000, C 0.000 }
gfCNCPoint3[29966] = {X 587.6457, Y 6.6169, Z -4.6667, A 0.000, B 0.000, C 0.000 }
gfCNCPoint3[29967] = {X 587.5870, Y 5.9340, Z -4.6667, A 0.000, B 0.000, C 0.000 }
